Yaskawa INFORM job: DEMO_ROOF_SIDE_0625_3PAINT_24.JBI

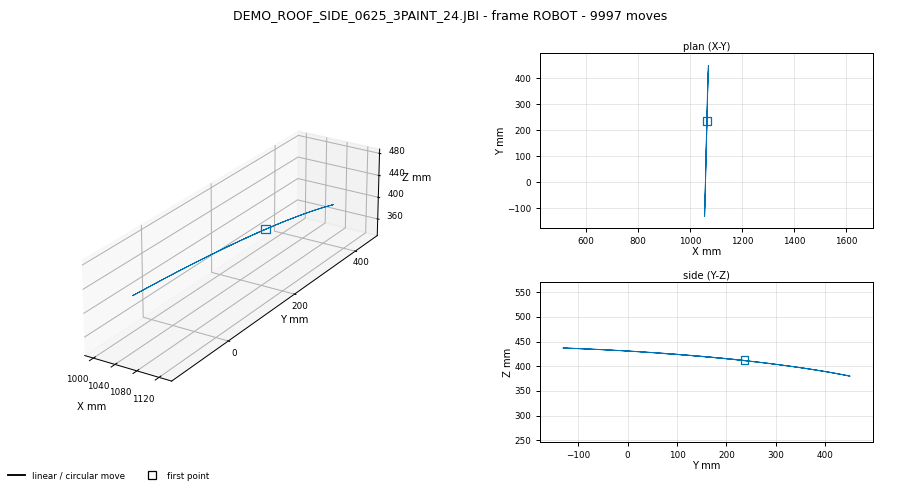
[picture p0: tool path of DEMO_ROOF_SIDE_0625_3PAINT_24.JBI in frame ROBOT, 9997 of 9997 moves have a stored position in this frame; points joined in program order, loops and branches not executed]
/JOB
//NAME DEMO_ROOF_SIDE_0625_3PAINT24
//POS
///NPOS 9997,0,0,0,0,0
///TOOL 0
///USER 0
///POSTYPE ROBOT
///RECTAN
///RCONF 1,0,0,0,0,0,0,0,0,0,0,0,0,0,0,0,0,0,0,0,0,0,0,0
C00000=1065.448,236.370,411.983,173.336,31.079,155.692
C00001=1065.443,236.150,412.007,173.335,31.075,155.691
C00002=1065.438,235.930,412.031,173.333,31.072,155.691
C00003=1065.433,235.710,412.055,173.331,31.069,155.690
C00004=1065.427,235.489,412.080,173.329,31.065,155.690
C00005=1065.422,235.270,412.102,173.326,31.062,155.689
C00006=1065.416,235.049,412.127,173.325,31.058,155.688
C00007=1065.411,234.830,412.151,173.323,31.055,155.688
C00008=1065.405,234.581,412.178,173.321,31.050,155.687
C00009=1065.399,234.332,412.204,173.318,31.047,155.686
C00010=1065.393,234.085,412.232,173.317,31.042,155.686
C00011=1065.388,233.835,412.259,173.314,31.038,155.685
C00012=1065.382,233.587,412.286,173.312,31.034,155.684
C00013=1065.376,233.339,412.313,173.309,31.030,155.683
C00014=1065.370,233.090,412.339,173.308,31.027,155.683
C00015=1065.364,232.842,412.367,173.305,31.022,155.682
C00016=1065.358,232.593,412.394,173.303,31.018,155.681
C00017=1065.352,232.345,412.420,173.300,31.015,155.681
C00018=1065.346,232.096,412.447,173.299,31.010,155.680
C00019=1065.340,231.848,412.474,173.296,31.006,155.679
C00020=1065.334,231.599,412.501,173.294,31.002,155.678
C00021=1065.328,231.350,412.528,173.293,30.998,155.678
C00022=1065.322,231.102,412.554,173.290,30.995,155.677
C00023=1065.316,230.853,412.581,173.288,30.990,155.676
C00024=1065.310,230.606,412.608,173.285,30.986,155.676
C00025=1065.304,230.357,412.635,173.284,30.982,155.675
C00026=1065.298,230.108,412.662,173.281,30.978,155.674
C00027=1065.292,229.860,412.689,173.279,30.975,155.674
C00028=1065.286,229.611,412.716,173.276,30.970,155.673
C00029=1065.280,229.363,412.742,173.275,30.966,155.672
C00030=1065.274,229.114,412.769,173.273,30.962,155.671
C00031=1065.268,228.866,412.794,173.270,30.958,155.671
C00032=1065.262,228.616,412.821,173.269,30.955,155.670
C00033=1065.256,228.368,412.848,173.266,30.950,155.669
C00034=1065.250,228.120,412.875,173.264,30.946,155.669
C00035=1065.244,227.871,412.902,173.261,30.943,155.668
C00036=1065.237,227.623,412.928,173.260,30.938,155.667
C00037=1065.232,227.374,412.954,173.258,30.935,155.667
C00038=1065.226,227.126,412.981,173.255,30.931,155.666
C00039=1065.220,226.878,413.008,173.253,30.926,155.665
C00040=1065.213,226.629,413.034,173.251,30.923,155.664
C00041=1065.207,226.380,413.060,173.249,30.919,155.664
C00042=1065.202,226.131,413.087,173.246,30.914,155.663
C00043=1065.196,225.883,413.113,173.245,30.911,155.662
C00044=1065.189,225.634,413.140,173.243,30.906,155.662
C00045=1065.183,225.386,413.166,173.240,30.903,155.661
C00046=1065.177,225.137,413.192,173.238,30.899,155.660
C00047=1065.172,224.889,413.219,173.236,30.894,155.659
C00048=1065.166,224.640,413.246,173.234,30.891,155.659
C00049=1065.159,224.392,413.272,173.232,30.886,155.658
C00050=1065.153,224.143,413.298,173.230,30.882,155.657
C00051=1065.148,223.894,413.325,173.228,30.878,155.657
C00052=1065.142,223.646,413.351,173.225,30.874,155.656
C00053=1065.135,223.398,413.377,173.223,30.870,155.655
C00054=1065.130,223.149,413.403,173.222,30.866,155.654
C00055=1065.124,222.900,413.430,173.219,30.862,155.654
C00056=1065.118,222.676,413.454,173.217,30.859,155.653
C00057=1065.113,222.452,413.477,173.215,30.855,155.652
C00058=1065.108,222.229,413.501,173.214,30.851,155.652
C00059=1065.102,222.004,413.525,173.212,30.848,155.651
C00060=1065.097,221.780,413.548,173.210,30.844,155.650
C00061=1065.092,221.556,413.572,173.208,30.841,155.650
C00062=1065.087,221.332,413.595,173.206,30.837,155.649
C00063=1065.080,221.108,413.619,173.204,30.833,155.649
C00064=1065.075,220.859,413.645,173.202,30.829,155.648
C00065=1065.069,220.611,413.671,173.200,30.825,155.647
C00066=1065.063,220.362,413.697,173.198,30.821,155.647
C00067=1065.057,220.114,413.723,173.196,30.817,155.646
C00068=1065.051,219.865,413.749,173.194,30.813,155.645
C00069=1065.044,219.616,413.775,173.192,30.809,155.644
C00070=1065.038,219.367,413.801,173.190,30.805,155.644
C00071=1065.032,219.119,413.827,173.187,30.801,155.643
C00072=1065.026,218.870,413.853,173.186,30.797,155.642
C00073=1065.020,218.622,413.879,173.184,30.793,155.642
C00074=1065.014,218.373,413.905,173.181,30.789,155.641
C00075=1065.008,218.125,413.931,173.180,30.785,155.640
C00076=1065.002,217.876,413.957,173.178,30.781,155.639
C00077=1064.996,217.628,413.983,173.175,30.777,155.639
C00078=1064.991,217.379,414.009,173.173,30.773,155.638
C00079=1064.984,217.131,414.034,173.172,30.769,155.637
C00080=1064.979,216.882,414.061,173.169,30.765,155.637
C00081=1064.972,216.634,414.086,173.167,30.760,155.636
C00082=1064.967,216.385,414.112,173.165,30.756,155.635
C00083=1064.960,216.137,414.138,173.163,30.752,155.634
C00084=1064.955,215.888,414.164,173.161,30.748,155.634
C00085=1064.949,215.639,414.190,173.160,30.744,155.633
C00086=1064.942,215.391,414.216,173.157,30.740,155.632
C00087=1064.937,215.142,414.242,173.155,30.736,155.631
C00088=1064.930,214.893,414.267,173.153,30.732,155.631
C00089=1064.925,214.645,414.294,173.151,30.728,155.630
C00090=1064.918,214.396,414.319,173.149,30.724,155.629
C00091=1064.913,214.147,414.345,173.147,30.720,155.629
C00092=1064.907,213.899,414.370,173.145,30.716,155.628
C00093=1064.900,213.651,414.396,173.143,30.712,155.627
C00094=1064.895,213.402,414.422,173.141,30.708,155.626
C00095=1064.889,213.153,414.448,173.139,30.703,155.626
C00096=1064.883,212.904,414.473,173.137,30.700,155.625
C00097=1064.877,212.655,414.499,173.135,30.695,155.624
C00098=1064.870,212.407,414.525,173.133,30.691,155.624
C00099=1064.864,212.159,414.550,173.131,30.687,155.623
C00100=1064.859,211.910,414.576,173.129,30.683,155.622
C00101=1064.853,211.662,414.601,173.127,30.679,155.621
C00102=1064.847,211.413,414.626,173.125,30.675,155.621
C00103=1064.842,211.164,414.652,173.123,30.671,155.620
C00104=1064.835,210.915,414.678,173.121,30.667,155.619
C00105=1064.829,210.667,414.703,173.119,30.663,155.619
C00106=1064.823,210.418,414.728,173.117,30.659,155.618
C00107=1064.817,210.169,414.754,173.115,30.655,155.617
C00108=1064.811,209.920,414.780,173.114,30.650,155.616
C00109=1064.805,209.672,414.805,173.111,30.646,155.616
C00110=1064.798,209.424,414.831,173.109,30.642,155.615
C00111=1064.792,209.175,414.856,173.108,30.638,155.614
C00112=1064.788,208.953,414.879,173.106,30.635,155.614
C00113=1064.782,208.732,414.901,173.104,30.631,155.613
C00114=1064.777,208.510,414.924,173.103,30.627,155.612
C00115=1064.771,208.288,414.947,173.101,30.624,155.612
C00116=1064.766,208.066,414.969,173.099,30.620,155.611
C00117=1064.761,207.845,414.992,173.097,30.616,155.610
C00118=1064.756,207.624,415.015,173.095,30.612,155.610
C00119=1064.750,207.401,415.037,173.093,30.609,155.609
C00120=1064.722,206.233,415.152,172.931,30.529,155.603
C00121=1064.714,205.844,415.190,172.928,30.523,155.602
C00122=1064.705,205.475,415.227,172.924,30.519,155.601
C00123=1064.696,205.104,415.263,172.922,30.514,155.601
C00124=1064.688,204.735,415.299,172.918,30.509,155.600
C00125=1064.679,204.365,415.336,172.915,30.504,155.599
C00126=1064.674,204.117,415.360,172.913,30.501,155.598
C00127=1064.668,203.867,415.385,172.910,30.498,155.598
C00128=1064.662,203.619,415.409,172.908,30.495,155.598
C00129=1064.656,203.370,415.434,172.906,30.492,155.597
C00130=1064.650,203.121,415.457,172.904,30.488,155.596
C00131=1064.645,202.873,415.482,172.901,30.485,155.596
C00132=1064.639,202.624,415.507,172.899,30.482,155.595
C00133=1064.634,202.375,415.531,172.897,30.479,155.595
C00134=1064.627,202.126,415.555,172.895,30.476,155.594
C00135=1064.622,201.878,415.579,172.892,30.472,155.594
C00136=1064.616,201.629,415.604,172.891,30.469,155.593
C00137=1064.610,201.380,415.628,172.888,30.466,155.593
C00138=1064.604,201.131,415.652,172.886,30.463,155.592
C00139=1064.598,200.883,415.676,172.883,30.460,155.592
C00140=1064.593,200.634,415.700,172.882,30.457,155.592
C00141=1064.586,200.385,415.724,172.880,30.454,155.591
C00142=1064.581,200.137,415.749,172.877,30.451,155.590
C00143=1064.574,199.888,415.773,172.875,30.448,155.590
C00144=1064.569,199.639,415.797,172.873,30.444,155.590
C00145=1064.562,199.390,415.821,172.871,30.441,155.589
C00146=1064.557,199.141,415.844,172.868,30.438,155.589
C00147=1064.551,198.893,415.868,172.867,30.435,155.588
C00148=1064.545,198.643,415.893,172.864,30.432,155.588
C00149=1064.539,198.395,415.916,172.862,30.429,155.587
C00150=1064.534,198.146,415.941,172.859,30.426,155.587
C00151=1064.527,197.897,415.965,172.858,30.423,155.586
C00152=1064.522,197.649,415.989,172.855,30.420,155.586
C00153=1064.515,197.400,416.013,172.853,30.417,155.585
C00154=1064.510,197.151,416.036,172.851,30.414,155.585
C00155=1064.504,196.902,416.060,172.849,30.411,155.584
C00156=1064.498,196.653,416.085,172.847,30.407,155.584
C00157=1064.492,196.405,416.108,172.844,30.405,155.583
C00158=1064.487,196.156,416.133,172.843,30.401,155.583
C00159=1064.481,195.907,416.156,172.840,30.398,155.582
C00160=1064.475,195.658,416.180,172.838,30.395,155.582
C00161=1064.469,195.410,416.204,172.836,30.392,155.581
C00162=1064.463,195.161,416.228,172.834,30.389,155.581
C00163=1064.458,194.912,416.251,172.832,30.386,155.580
C00164=1064.452,194.663,416.275,172.829,30.383,155.580
C00165=1064.446,194.415,416.299,172.827,30.380,155.579
C00166=1064.440,194.165,416.323,172.826,30.377,155.579
C00167=1064.435,193.917,416.347,172.823,30.373,155.578
C00168=1064.429,193.668,416.371,172.821,30.371,155.578
C00169=1064.423,193.419,416.394,172.819,30.367,155.577
C00170=1064.417,193.170,416.418,172.817,30.365,155.577
C00171=1064.411,192.922,416.442,172.815,30.362,155.576
C00172=1064.406,192.673,416.465,172.812,30.358,155.576
C00173=1064.400,192.424,416.489,172.811,30.355,155.576
C00174=1064.394,192.175,416.514,172.808,30.352,155.575
C00175=1064.388,191.926,416.537,172.806,30.349,155.574
C00176=1064.382,191.678,416.560,172.805,30.346,155.574
C00177=1064.377,191.429,416.584,172.802,30.343,155.574
C00178=1064.370,191.146,416.611,172.799,30.339,155.573
C00179=1064.364,190.863,416.638,172.797,30.336,155.572
C00180=1064.357,190.580,416.665,172.795,30.332,155.572
C00181=1064.351,190.297,416.692,172.792,30.329,155.571
C00182=1064.345,190.048,416.715,172.790,30.326,155.571
C00183=1064.340,189.799,416.739,172.789,30.323,155.570
C00184=1064.334,189.551,416.763,172.786,30.320,155.570
C00185=1064.328,189.301,416.786,172.784,30.317,155.569
C00186=1064.322,189.053,416.810,172.783,30.314,155.569
C00187=1064.316,188.804,416.833,172.780,30.311,155.569
C00188=1064.311,188.555,416.857,172.778,30.308,155.568
C00189=1064.305,188.306,416.880,172.776,30.304,155.567
C00190=1064.299,188.058,416.904,172.774,30.302,155.567
C00191=1064.294,187.809,416.927,172.772,30.298,155.567
C00192=1064.289,187.560,416.950,172.769,30.295,155.566
C00193=1064.282,187.311,416.974,172.767,30.292,155.566
C00194=1064.277,187.062,416.998,172.766,30.289,155.565
C00195=1064.271,186.814,417.022,172.763,30.286,155.565
C00196=1064.266,186.564,417.045,172.761,30.283,155.564
C00197=1064.260,186.315,417.068,172.760,30.280,155.564
C00198=1064.254,186.067,417.092,172.757,30.277,155.563
C00199=1064.249,185.818,417.115,172.755,30.274,155.563
C00200=1064.243,185.569,417.138,172.753,30.271,155.562
C00201=1064.237,185.321,417.162,172.752,30.268,155.562
C00202=1064.232,185.072,417.185,172.749,30.264,155.561
C00203=1064.227,184.823,417.208,172.747,30.262,155.561
C00204=1064.221,184.574,417.231,172.746,30.259,155.560
C00205=1064.214,184.325,417.255,172.743,30.256,155.560
C00206=1064.209,184.076,417.278,172.741,30.253,155.559
C00207=1064.203,183.827,417.301,172.739,30.250,155.559
C00208=1064.197,183.578,417.324,172.737,30.247,155.559
C00209=1064.191,183.330,417.348,172.735,30.244,155.558
C00210=1064.185,183.081,417.371,172.733,30.241,155.558
C00211=1064.179,182.831,417.394,172.731,30.238,155.557
C00212=1064.173,182.583,417.416,172.729,30.236,155.557
C00213=1064.167,182.334,417.439,172.727,30.232,155.556
C00214=1064.161,182.085,417.462,172.724,30.230,155.556
C00215=1064.155,181.836,417.485,172.723,30.227,155.555
C00216=1064.149,181.588,417.509,172.721,30.224,155.555
C00217=1064.144,181.339,417.532,172.718,30.221,155.554
C00218=1064.137,181.089,417.555,172.716,30.218,155.554
C00219=1064.131,180.841,417.578,172.715,30.215,155.554
C00220=1064.125,180.592,417.601,172.712,30.212,155.553
C00221=1064.119,180.343,417.623,172.710,30.209,155.553
C00222=1064.114,180.094,417.646,172.709,30.206,155.552
C00223=1064.108,179.845,417.669,172.706,30.203,155.552
C00224=1064.102,179.596,417.692,172.704,30.201,155.551
C00225=1064.096,179.347,417.715,172.702,30.198,155.551
C00226=1064.090,179.099,417.738,172.701,30.195,155.550
C00227=1064.084,178.850,417.761,172.698,30.192,155.550
C00228=1064.079,178.601,417.783,172.696,30.189,155.550
C00229=1064.073,178.352,417.806,172.695,30.186,155.549
C00230=1064.067,178.103,417.829,172.692,30.183,155.549
C00231=1064.061,177.854,417.852,172.690,30.180,155.548
C00232=1064.055,177.606,417.875,172.688,30.177,155.548
C00233=1064.049,177.357,417.898,172.687,30.175,155.547
C00234=1064.043,177.108,417.921,172.684,30.171,155.547
C00235=1064.038,176.859,417.944,172.682,30.169,155.546
C00236=1064.032,176.610,417.966,172.680,30.166,155.546
C00237=1064.025,176.362,417.989,172.679,30.163,155.545
C00238=1064.020,176.113,418.012,172.676,30.160,155.545
C00239=1064.014,175.864,418.035,172.674,30.157,155.545
C00240=1064.009,175.614,418.057,172.673,30.154,155.544
C00241=1064.003,175.365,418.080,172.670,30.151,155.544
C00242=1063.996,175.081,418.106,172.668,30.148,155.543
C00243=1063.989,174.798,418.132,172.666,30.144,155.543
C00244=1063.982,174.515,418.157,172.664,30.141,155.542
C00245=1063.975,174.232,418.183,172.661,30.138,155.542
C00246=1063.970,173.983,418.206,172.659,30.135,155.541
C00247=1063.964,173.734,418.229,172.658,30.132,155.541
C00248=1063.958,173.485,418.252,172.655,30.129,155.540
C00249=1063.953,173.236,418.274,172.653,30.126,155.540
C00250=1063.946,172.987,418.296,172.652,30.124,155.539
C00251=1063.941,172.739,418.319,172.650,30.120,155.539
C00252=1063.935,172.490,418.342,172.648,30.118,155.539
C00253=1063.930,172.240,418.364,172.645,30.115,155.538
C00254=1063.924,171.992,418.387,172.644,30.112,155.538
C00255=1063.918,171.743,418.410,172.642,30.109,155.537
C00256=1063.912,171.494,418.432,172.640,30.106,155.537
C00257=1063.907,171.245,418.455,172.638,30.103,155.536
C00258=1063.900,170.996,418.477,172.636,30.100,155.536
C00259=1063.895,170.747,418.500,172.634,30.098,155.535
C00260=1063.890,170.498,418.522,172.632,30.094,155.535
C00261=1063.884,170.249,418.545,172.631,30.092,155.534
C00262=1063.877,170.001,418.567,172.628,30.089,155.534
C00263=1063.872,169.751,418.589,172.626,30.086,155.534
C00264=1063.866,169.502,418.612,172.625,30.083,155.533
C00265=1063.860,169.254,418.635,172.623,30.080,155.533
C00266=1063.855,169.005,418.657,172.621,30.077,155.532
C00267=1063.849,168.756,418.679,172.618,30.074,155.532
C00268=1063.844,168.507,418.702,172.617,30.071,155.531
C00269=1063.837,168.258,418.724,172.615,30.068,155.531
C00270=1063.832,168.009,418.747,172.613,30.066,155.530
C00271=1063.827,167.760,418.769,172.612,30.063,155.530
C00272=1063.820,167.512,418.791,172.609,30.059,155.530
C00273=1063.815,167.262,418.813,172.607,30.057,155.529
C00274=1063.809,167.013,418.836,172.605,30.054,155.529
C00275=1063.804,166.764,418.859,172.604,30.051,155.528
C00276=1063.798,166.516,418.881,172.602,30.048,155.528
C00277=1063.793,166.266,418.903,172.599,30.045,155.527
C00278=1063.787,166.017,418.926,172.598,30.042,155.527
C00279=1063.781,165.768,418.947,172.596,30.039,155.526
C00280=1063.775,165.520,418.970,172.594,30.036,155.526
C00281=1063.770,165.271,418.992,172.592,30.033,155.525
C00282=1063.764,165.022,419.015,172.591,30.031,155.525
C00283=1063.758,164.772,419.037,172.588,30.027,155.525
C00284=1063.753,164.524,419.059,172.586,30.025,155.524
C00285=1063.747,164.275,419.081,172.585,30.022,155.524
C00286=1063.741,164.025,419.103,172.583,30.019,155.523
C00287=1063.736,163.777,419.126,172.581,30.016,155.523
C00288=1063.730,163.528,419.147,172.580,30.013,155.522
C00289=1063.724,163.279,419.170,172.577,30.010,155.522
C00290=1063.720,163.030,419.192,172.575,30.007,155.521
C00291=1063.713,162.781,419.214,172.573,30.004,155.521
C00292=1063.708,162.532,419.237,172.572,30.001,155.521
C00293=1063.703,162.283,419.259,172.570,29.999,155.520
C00294=1063.696,162.035,419.281,172.568,29.995,155.520
C00295=1063.691,161.785,419.303,172.567,29.993,155.519
C00296=1063.686,161.537,419.325,172.564,29.990,155.519
C00297=1063.680,161.288,419.348,172.562,29.987,155.518
C00298=1063.674,161.038,419.370,172.560,29.984,155.518
C00299=1063.668,160.789,419.391,172.559,29.981,155.517
C00300=1063.663,160.541,419.413,172.557,29.978,155.517
C00301=1063.657,160.292,419.436,172.555,29.975,155.516
C00302=1063.651,160.043,419.457,172.554,29.973,155.516
C00303=1063.645,159.794,419.479,172.551,29.970,155.516
C00304=1063.640,159.545,419.501,172.549,29.967,155.515
C00305=1063.634,159.295,419.522,172.548,29.964,155.515
C00306=1063.626,159.012,419.547,172.546,29.961,155.514
C00307=1063.620,158.728,419.572,172.543,29.958,155.514
C00308=1063.613,158.445,419.597,172.542,29.955,155.513
C00309=1063.607,158.161,419.622,172.539,29.952,155.513
C00310=1063.601,157.912,419.644,172.537,29.948,155.512
C00311=1063.596,157.663,419.666,172.535,29.946,155.512
C00312=1063.590,157.414,419.688,172.534,29.943,155.512
C00313=1063.584,157.165,419.709,172.532,29.940,155.511
C00314=1063.578,156.916,419.730,172.530,29.938,155.511
C00315=1063.573,156.667,419.753,172.529,29.934,155.510
C00316=1063.566,156.418,419.775,172.526,29.932,155.510
C00317=1063.561,156.170,419.796,172.524,29.929,155.509
C00318=1063.554,155.920,419.818,172.522,29.926,155.509
C00319=1063.549,155.671,419.840,172.521,29.923,155.509
C00320=1063.543,155.422,419.861,172.519,29.920,155.508
C00321=1063.537,155.173,419.883,172.517,29.918,155.508
C00322=1063.531,154.924,419.905,172.516,29.915,155.507
C00323=1063.526,154.675,419.927,172.514,29.912,155.507
C00324=1063.520,154.426,419.948,172.512,29.909,155.506
C00325=1063.514,154.177,419.970,172.509,29.907,155.506
C00326=1063.508,153.928,419.991,172.508,29.903,155.505
C00327=1063.502,153.679,420.013,172.506,29.901,155.505
C00328=1063.497,153.430,420.034,172.504,29.898,155.505
C00329=1063.490,153.181,420.056,172.503,29.895,155.504
C00330=1063.485,152.932,420.078,172.501,29.893,155.504
C00331=1063.480,152.683,420.099,172.499,29.890,155.503
C00332=1063.473,152.434,420.121,172.498,29.887,155.503
C00333=1063.468,152.186,420.142,172.496,29.884,155.502
C00334=1063.462,151.936,420.164,172.494,29.881,155.502
C00335=1063.456,151.686,420.185,172.491,29.878,155.502
C00336=1063.450,151.438,420.206,172.490,29.876,155.501
C00337=1063.445,151.188,420.228,172.488,29.873,155.501
C00338=1063.439,150.940,420.249,172.486,29.870,155.500
C00339=1063.433,150.691,420.271,172.485,29.867,155.500
C00340=1063.427,150.442,420.292,172.483,29.864,155.499
C00341=1063.421,150.193,420.314,172.481,29.862,155.499
C00342=1063.415,149.944,420.336,172.479,29.859,155.499
C00343=1063.410,149.695,420.356,172.478,29.856,155.498
C00344=1063.404,149.445,420.378,172.476,29.854,155.498
C00345=1063.398,149.197,420.399,172.474,29.851,155.497
C00346=1063.392,148.948,420.421,172.473,29.848,155.497
C00347=1063.386,148.699,420.442,172.471,29.845,155.496
C00348=1063.381,148.449,420.463,172.468,29.842,155.496
C00349=1063.375,148.201,420.484,172.467,29.839,155.496
C00350=1063.369,147.952,420.506,172.465,29.837,155.495
C00351=1063.363,147.703,420.527,172.463,29.834,155.495
C00352=1063.357,147.453,420.548,172.461,29.831,155.494
C00353=1063.351,147.204,420.570,172.460,29.829,155.494
C00354=1063.346,146.956,420.591,172.458,29.826,155.494
C00355=1063.340,146.707,420.613,172.456,29.823,155.493
C00356=1063.334,146.457,420.633,172.455,29.820,155.493
C00357=1063.328,146.208,420.655,172.453,29.817,155.492
C00358=1063.323,145.960,420.676,172.451,29.815,155.492
C00359=1063.317,145.710,420.697,172.449,29.812,155.491
C00360=1063.310,145.462,420.718,172.448,29.809,155.491
C00361=1063.304,145.212,420.739,172.446,29.806,155.491
C00362=1063.299,144.963,420.760,172.444,29.804,155.490
C00363=1063.293,144.714,420.781,172.442,29.801,155.490
C00364=1063.287,144.466,420.803,172.440,29.798,155.489
C00365=1063.281,144.216,420.824,172.438,29.795,155.489
C00366=1063.276,143.967,420.845,172.437,29.792,155.489
C00367=1063.270,143.717,420.866,172.435,29.790,155.488
C00368=1063.264,143.469,420.886,172.433,29.787,155.488
C00369=1063.258,143.220,420.908,172.431,29.784,155.487
C00370=1063.251,142.937,420.932,172.430,29.781,155.487
C00371=1063.245,142.653,420.956,172.428,29.778,155.486
C00372=1063.238,142.369,420.980,172.426,29.775,155.486
C00373=1063.231,142.085,421.004,172.424,29.771,155.485
C00374=1063.225,141.835,421.025,172.422,29.769,155.485
C00375=1063.220,141.586,421.046,172.420,29.766,155.485
C00376=1063.215,141.337,421.066,172.419,29.763,155.484
C00377=1063.208,141.088,421.088,172.417,29.761,155.484
C00378=1063.203,140.839,421.109,172.415,29.758,155.483
C00379=1063.196,140.590,421.130,172.414,29.755,155.483
C00380=1063.191,140.341,421.150,172.412,29.753,155.482
C00381=1063.185,140.092,421.172,172.410,29.750,155.482
C00382=1063.180,139.842,421.192,172.408,29.747,155.482
C00383=1063.174,139.593,421.213,172.407,29.744,155.481
C00384=1063.167,139.344,421.234,172.405,29.741,155.481
C00385=1063.162,139.095,421.255,172.403,29.738,155.480
C00386=1063.156,138.846,421.276,172.402,29.736,155.480
C00387=1063.150,138.597,421.296,172.400,29.733,155.479
C00388=1063.145,138.348,421.317,172.398,29.730,155.479
C00389=1063.139,138.099,421.338,172.397,29.728,155.479
C00390=1063.133,137.850,421.358,172.395,29.725,155.478
C00391=1063.126,137.601,421.380,172.393,29.722,155.478
C00392=1063.121,137.352,421.401,172.391,29.719,155.477
C00393=1063.115,137.103,421.420,172.389,29.717,155.477
C00394=1063.109,136.854,421.442,172.387,29.714,155.477
C00395=1063.104,136.605,421.463,172.385,29.711,155.476
C00396=1063.097,136.355,421.483,172.384,29.709,155.476
C00397=1063.092,136.107,421.504,172.382,29.706,155.475
C00398=1063.086,135.858,421.524,172.380,29.703,155.475
C00399=1063.080,135.608,421.545,172.379,29.700,155.475
C00400=1063.074,135.359,421.566,172.377,29.698,155.474
C00401=1063.068,135.111,421.586,172.375,29.695,155.474
C00402=1063.062,134.861,421.607,172.374,29.692,155.473
C00403=1063.056,134.612,421.627,172.372,29.689,155.473
C00404=1063.051,134.364,421.649,172.370,29.686,155.472
C00405=1063.045,134.114,421.669,172.368,29.684,155.472
C00406=1063.039,133.865,421.689,172.367,29.681,155.472
C00407=1063.034,133.616,421.710,172.365,29.678,155.471
C00408=1063.027,133.366,421.730,172.363,29.676,155.471
C00409=1063.022,133.118,421.752,172.363,29.673,155.470
C00410=1063.016,132.869,421.772,172.361,29.670,155.470
C00411=1063.010,132.619,421.792,172.359,29.668,155.470
C00412=1063.004,132.370,421.813,172.358,29.665,155.469
C00413=1062.998,132.121,421.833,172.356,29.662,155.469
C00414=1062.993,131.873,421.854,172.354,29.659,155.468
C00415=1062.986,131.623,421.875,172.352,29.657,155.468
C00416=1062.981,131.374,421.895,172.351,29.654,155.468
C00417=1062.974,131.125,421.915,172.349,29.651,155.467
C00418=1062.968,130.876,421.935,172.347,29.649,155.467
C00419=1062.963,130.627,421.956,172.346,29.646,155.466
C00420=1062.957,130.377,421.976,172.344,29.643,155.466
C00421=1062.951,130.128,421.996,172.342,29.641,155.465
C00422=1062.945,129.879,422.017,172.341,29.638,155.465
C00423=1062.939,129.630,422.037,172.339,29.635,155.465
C00424=1062.933,129.381,422.057,172.337,29.632,155.464
C00425=1062.928,129.132,422.078,172.335,29.630,155.464
C00426=1062.921,128.883,422.098,172.334,29.627,155.463
C00427=1062.915,128.634,422.119,172.332,29.624,155.463
C00428=1062.909,128.385,422.139,172.330,29.622,155.463
C00429=1062.903,128.136,422.159,172.329,29.619,155.462
C00430=1062.897,127.887,422.179,172.327,29.617,155.462
C00431=1062.891,127.638,422.199,172.325,29.614,155.462
C00432=1062.886,127.389,422.220,172.324,29.611,155.461
C00433=1062.880,127.140,422.240,172.322,29.609,155.461
C00434=1062.872,126.855,422.263,172.320,29.605,155.460
C00435=1062.866,126.571,422.286,172.318,29.602,155.460
C00436=1062.859,126.286,422.309,172.316,29.599,155.459
C00437=1062.853,126.003,422.332,172.314,29.596,155.459
C00438=1062.846,125.753,422.352,172.313,29.594,155.458
C00439=1062.840,125.504,422.372,172.311,29.591,155.458
C00440=1062.835,125.255,422.392,172.309,29.588,155.458
C00441=1062.829,125.006,422.412,172.307,29.586,155.457
C00442=1062.823,124.757,422.433,172.306,29.583,155.457
C00443=1062.817,124.508,422.453,172.304,29.580,155.456
C00444=1062.811,124.259,422.473,172.302,29.577,155.456
C00445=1062.805,124.010,422.493,172.301,29.575,155.456
C00446=1062.799,123.761,422.513,172.299,29.572,155.455
C00447=1062.793,123.511,422.533,172.297,29.569,155.455
C00448=1062.788,123.262,422.553,172.297,29.567,155.454
C00449=1062.782,123.013,422.573,172.295,29.564,155.454
C00450=1062.776,122.764,422.593,172.293,29.561,155.454
C00451=1062.770,122.515,422.613,172.292,29.559,155.453
C00452=1062.765,122.266,422.634,172.290,29.556,155.453
C00453=1062.758,122.016,422.653,172.288,29.553,155.452
C00454=1062.752,121.767,422.673,172.287,29.550,155.452
C00455=1062.746,121.518,422.693,172.285,29.548,155.452
C00456=1062.741,121.269,422.714,172.283,29.544,155.451
C00457=1062.735,121.020,422.733,172.281,29.542,155.451
C00458=1062.729,120.771,422.753,172.280,29.539,155.450
C00459=1062.723,120.522,422.773,172.278,29.536,155.450
C00460=1062.718,120.272,422.794,172.276,29.534,155.449
C00461=1062.712,120.023,422.813,172.275,29.531,155.449
C00462=1062.706,119.774,422.833,172.273,29.528,155.449
C00463=1062.700,119.525,422.853,172.272,29.526,155.448
C00464=1062.694,119.277,422.873,172.271,29.523,155.448
C00465=1062.689,119.027,422.893,172.269,29.520,155.447
C00466=1062.683,118.778,422.913,172.267,29.517,155.447
C00467=1062.677,118.529,422.933,172.266,29.515,155.447
C00468=1062.671,118.280,422.952,172.264,29.512,155.446
C00469=1062.665,118.031,422.972,172.262,29.509,155.446
C00470=1062.659,117.781,422.993,172.261,29.507,155.445
C00471=1062.654,117.532,423.012,172.259,29.504,155.445
C00472=1062.648,117.283,423.032,172.257,29.501,155.444
C00473=1062.642,117.033,423.051,172.256,29.498,155.444
C00474=1062.636,116.785,423.071,172.254,29.496,155.444
C00475=1062.631,116.536,423.092,172.253,29.493,155.443
C00476=1062.625,116.286,423.111,172.251,29.490,155.443
C00477=1062.619,116.037,423.131,172.250,29.488,155.442
C00478=1062.613,115.788,423.150,172.248,29.484,155.442
C00479=1062.607,115.539,423.170,172.246,29.482,155.441
C00480=1062.602,115.290,423.191,172.245,29.479,155.441
C00481=1062.596,115.040,423.210,172.243,29.476,155.441
C00482=1062.590,114.792,423.230,172.241,29.474,155.440
C00483=1062.585,114.542,423.249,172.240,29.471,155.440
C00484=1062.579,114.293,423.269,172.238,29.468,155.439
C00485=1062.573,114.044,423.288,172.236,29.465,155.439
C00486=1062.567,113.795,423.308,172.236,29.463,155.439
C00487=1062.561,113.546,423.328,172.234,29.460,155.438
C00488=1062.555,113.297,423.348,172.232,29.457,155.438
C00489=1062.550,113.048,423.367,172.231,29.455,155.437
C00490=1062.544,112.799,423.387,172.229,29.452,155.437
C00491=1062.538,112.549,423.406,172.227,29.449,155.437
C00492=1062.531,112.300,423.426,172.226,29.446,155.436
C00493=1062.526,112.050,423.446,172.224,29.444,155.436
C00494=1062.520,111.801,423.465,172.222,29.441,155.435
C00495=1062.514,111.552,423.485,172.221,29.438,155.435
C00496=1062.508,111.303,423.504,172.220,29.436,155.435
C00497=1062.502,111.054,423.524,172.218,29.433,155.434
C00498=1062.496,110.770,423.546,172.215,29.430,155.434
C00499=1062.488,110.485,423.568,172.214,29.427,155.433
C00500=1062.482,110.201,423.589,172.212,29.424,155.433
C00501=1062.475,109.917,423.612,172.211,29.421,155.432
C00502=1062.469,109.667,423.631,172.209,29.419,155.432
C00503=1062.463,109.419,423.651,172.207,29.416,155.432
C00504=1062.457,109.169,423.670,172.205,29.413,155.431
C00505=1062.451,108.920,423.689,172.204,29.410,155.431
C00506=1062.445,108.671,423.709,172.203,29.408,155.430
C00507=1062.439,108.422,423.728,172.201,29.405,155.430
C00508=1062.434,108.172,423.747,172.200,29.402,155.430
C00509=1062.428,107.924,423.767,172.198,29.400,155.429
C00510=1062.421,107.674,423.786,172.196,29.397,155.429
C00511=1062.416,107.425,423.805,172.195,29.394,155.428
C00512=1062.410,107.176,423.825,172.193,29.392,155.428
C00513=1062.404,106.927,423.845,172.191,29.389,155.428
C00514=1062.398,106.677,423.864,172.190,29.386,155.427
C00515=1062.392,106.428,423.882,172.189,29.384,155.427
C00516=1062.386,106.179,423.902,172.187,29.381,155.426
C00517=1062.381,105.931,423.921,172.186,29.378,155.426
C00518=1062.375,105.681,423.941,172.184,29.375,155.426
C00519=1062.369,105.432,423.959,172.182,29.373,155.425
C00520=1062.363,105.183,423.978,172.181,29.370,155.425
C00521=1062.357,104.933,423.998,172.179,29.368,155.424
C00522=1062.351,104.684,424.018,172.177,29.365,155.424
C00523=1062.345,104.435,424.036,172.176,29.362,155.424
C00524=1062.339,104.186,424.056,172.175,29.360,155.423
C00525=1062.333,103.936,424.075,172.173,29.357,155.423
C00526=1062.328,103.687,424.094,172.172,29.354,155.422
C00527=1062.321,103.438,424.113,172.170,29.352,155.422
C00528=1062.315,103.189,424.133,172.168,29.349,155.422
C00529=1062.310,102.940,424.152,172.167,29.346,155.421
C00530=1062.305,102.691,424.171,172.165,29.343,155.421
C00531=1062.298,102.442,424.189,172.164,29.341,155.420
C00532=1062.292,102.192,424.209,172.162,29.338,155.420
C00533=1062.287,101.943,424.228,172.161,29.335,155.420
C00534=1062.281,101.693,424.247,172.159,29.333,155.419
C00535=1062.275,101.444,424.266,172.157,29.330,155.419
C00536=1062.269,101.195,424.285,172.156,29.327,155.418
C00537=1062.263,100.945,424.304,172.154,29.324,155.418
C00538=1062.257,100.697,424.323,172.152,29.322,155.418
C00539=1062.252,100.448,424.342,172.152,29.319,155.417
C00540=1062.245,100.199,424.360,172.150,29.316,155.417
C00541=1062.240,99.949,424.380,172.148,29.314,155.416
C00542=1062.233,99.700,424.398,172.147,29.311,155.416
C00543=1062.228,99.451,424.418,172.145,29.309,155.416
C00544=1062.221,99.201,424.436,172.143,29.306,155.415
C00545=1062.215,98.952,424.455,172.142,29.303,155.415
C00546=1062.209,98.703,424.474,172.141,29.301,155.414
C00547=1062.204,98.454,424.493,172.139,29.298,155.414
C00548=1062.197,98.205,424.512,172.138,29.295,155.414
C00549=1062.192,97.956,424.531,172.136,29.293,155.413
C00550=1062.185,97.706,424.550,172.134,29.290,155.413
C00551=1062.180,97.457,424.569,172.133,29.287,155.412
C00552=1062.173,97.208,424.587,172.131,29.284,155.412
C00553=1062.168,96.958,424.607,172.129,29.282,155.412
C00554=1062.162,96.710,424.625,172.129,29.280,155.411
C00555=1062.156,96.461,424.644,172.127,29.277,155.411
C00556=1062.150,96.212,424.663,172.125,29.274,155.410
C00557=1062.144,95.961,424.681,172.124,29.271,155.410
C00558=1062.138,95.712,424.700,172.122,29.269,155.410
C00559=1062.132,95.463,424.719,172.120,29.266,155.409
C00560=1062.126,95.214,424.738,172.120,29.263,155.409
C00561=1062.121,94.965,424.757,172.118,29.261,155.408
C00562=1062.114,94.681,424.778,172.116,29.258,155.408
C00563=1062.107,94.396,424.800,172.114,29.254,155.407
C00564=1062.100,94.112,424.821,172.112,29.252,155.407
C00565=1062.094,93.828,424.842,172.110,29.248,155.407
C00566=1062.087,93.579,424.861,172.109,29.246,155.406
C00567=1062.082,93.330,424.879,172.108,29.243,155.406
C00568=1062.076,93.080,424.898,172.106,29.240,155.405
C00569=1062.069,92.831,424.916,172.105,29.238,155.405
C00570=1062.064,92.582,424.936,172.103,29.235,155.405
C00571=1062.058,92.333,424.954,172.101,29.233,155.404
C00572=1062.053,92.083,424.973,172.100,29.230,155.404
C00573=1062.046,91.834,424.991,172.098,29.227,155.403
C00574=1062.040,91.585,425.010,172.097,29.225,155.403
C00575=1062.035,91.336,425.029,172.096,29.222,155.403
C00576=1062.029,91.087,425.047,172.094,29.219,155.402
C00577=1062.023,90.837,425.066,172.092,29.216,155.402
C00578=1062.016,90.588,425.085,172.091,29.214,155.401
C00579=1062.011,90.339,425.102,172.089,29.211,155.401
C00580=1062.005,90.089,425.121,172.088,29.208,155.401
C00581=1061.999,89.840,425.140,172.087,29.206,155.400
C00582=1061.993,89.591,425.158,172.085,29.203,155.400
C00583=1061.987,89.342,425.176,172.083,29.201,155.399
C00584=1061.981,89.093,425.195,172.082,29.198,155.399
C00585=1061.975,88.843,425.213,172.080,29.195,155.399
C00586=1061.969,88.594,425.232,172.079,29.193,155.398
C00587=1061.963,88.345,425.250,172.078,29.190,155.398
C00588=1061.957,88.096,425.268,172.076,29.187,155.397
C00589=1061.951,87.846,425.287,172.074,29.185,155.397
C00590=1061.945,87.597,425.305,172.073,29.182,155.397
C00591=1061.939,87.348,425.324,172.071,29.180,155.396
C00592=1061.933,87.098,425.342,172.069,29.177,155.396
C00593=1061.926,86.849,425.360,172.069,29.174,155.396
C00594=1061.921,86.600,425.380,172.067,29.172,155.395
C00595=1061.915,86.351,425.397,172.065,29.169,155.395
C00596=1061.909,86.102,425.416,172.064,29.166,155.394
C00597=1061.903,85.852,425.434,172.062,29.164,155.394
C00598=1061.897,85.604,425.452,172.060,29.161,155.394
C00599=1061.891,85.354,425.470,172.060,29.159,155.393
C00600=1061.885,85.104,425.489,172.058,29.156,155.393
C00601=1061.880,84.855,425.507,172.056,29.153,155.392
C00602=1061.873,84.606,425.525,172.055,29.150,155.392
C00603=1061.867,84.356,425.543,172.053,29.148,155.392
C00604=1061.861,84.108,425.562,172.051,29.145,155.391
C00605=1061.855,83.858,425.580,172.051,29.143,155.391
C00606=1061.849,83.609,425.599,172.049,29.140,155.390
C00607=1061.844,83.360,425.616,172.047,29.137,155.390
C00608=1061.838,83.110,425.634,172.046,29.135,155.390
C00609=1061.831,82.861,425.653,172.044,29.132,155.389
C00610=1061.826,82.612,425.670,172.042,29.129,155.389
C00611=1061.819,82.363,425.689,172.042,29.127,155.388
C00612=1061.813,82.113,425.707,172.040,29.124,155.388
C00613=1061.808,81.864,425.726,172.038,29.121,155.388
C00614=1061.802,81.615,425.744,172.037,29.118,155.387
C00615=1061.797,81.366,425.761,172.035,29.116,155.387
C00616=1061.790,81.116,425.780,172.034,29.114,155.387
C00617=1061.784,80.867,425.798,172.033,29.111,155.386
C00618=1061.778,80.618,425.816,172.031,29.108,155.386
C00619=1061.772,80.369,425.834,172.029,29.105,155.385
C00620=1061.767,80.119,425.852,172.028,29.103,155.385
C00621=1061.761,79.870,425.871,172.026,29.100,155.385
C00622=1061.755,79.620,425.889,172.025,29.097,155.384
C00623=1061.749,79.371,425.907,172.024,29.095,155.384
C00624=1061.743,79.122,425.925,172.022,29.092,155.383
C00625=1061.737,78.873,425.943,172.020,29.089,155.383
C00626=1061.731,78.589,425.963,172.019,29.086,155.383
C00627=1061.724,78.305,425.984,172.017,29.083,155.382
C00628=1061.717,78.020,426.004,172.016,29.080,155.382
C00629=1061.710,77.735,426.025,172.014,29.077,155.381
C00630=1061.704,77.486,426.043,172.012,29.075,155.381
C00631=1061.698,77.237,426.061,172.011,29.072,155.380
C00632=1061.691,76.988,426.078,172.009,29.069,155.380
C00633=1061.686,76.739,426.096,172.008,29.067,155.380
C00634=1061.680,76.490,426.114,172.007,29.064,155.379
C00635=1061.674,76.241,426.132,172.005,29.062,155.379
C00636=1061.668,75.991,426.150,172.003,29.059,155.379
C00637=1061.662,75.741,426.168,172.002,29.056,155.378
C00638=1061.656,75.492,426.185,172.000,29.053,155.378
C00639=1061.650,75.243,426.204,171.999,29.051,155.377
C00640=1061.644,74.994,426.222,171.998,29.048,155.377
C00641=1061.638,74.744,426.240,171.996,29.046,155.377
C00642=1061.632,74.495,426.257,171.994,29.043,155.376
C00643=1061.626,74.246,426.274,171.993,29.040,155.376
C00644=1061.620,73.996,426.292,171.992,29.038,155.375
C00645=1061.614,73.747,426.310,171.990,29.035,155.375
C00646=1061.608,73.498,426.329,171.989,29.032,155.375
C00647=1061.602,73.249,426.346,171.987,29.030,155.374
C00648=1061.596,72.999,426.364,171.985,29.027,155.374
C00649=1061.590,72.750,426.381,171.984,29.025,155.374
C00650=1061.584,72.501,426.399,171.983,29.022,155.373
C00651=1061.578,72.251,426.417,171.981,29.019,155.373
C00652=1061.572,72.002,426.435,171.980,29.017,155.372
C00653=1061.567,71.753,426.452,171.978,29.014,155.372
C00654=1061.560,71.503,426.470,171.976,29.012,155.372
C00655=1061.555,71.254,426.488,171.976,29.009,155.371
C00656=1061.548,71.004,426.505,171.974,29.006,155.371
C00657=1061.543,70.755,426.523,171.972,29.004,155.370
C00658=1061.536,70.506,426.540,171.971,29.001,155.370
C00659=1061.531,70.257,426.558,171.969,28.998,155.370
C00660=1061.525,70.007,426.576,171.969,28.996,155.369
C00661=1061.519,69.758,426.593,171.967,28.993,155.369
C00662=1061.512,69.508,426.611,171.965,28.991,155.368
C00663=1061.507,69.259,426.628,171.964,28.988,155.368
C00664=1061.501,69.010,426.646,171.962,28.985,155.368
C00665=1061.495,68.761,426.663,171.960,28.982,155.367
C00666=1061.489,68.512,426.681,171.960,28.980,155.367
C00667=1061.483,68.262,426.699,171.958,28.978,155.367
C00668=1061.477,68.013,426.716,171.956,28.975,155.366
C00669=1061.471,67.764,426.734,171.955,28.972,155.366
C00670=1061.465,67.515,426.751,171.953,28.969,155.365
C00671=1061.458,67.265,426.769,171.952,28.967,155.365
C00672=1061.453,67.016,426.786,171.951,28.965,155.365
C00673=1061.446,66.766,426.804,171.949,28.962,155.364
C00674=1061.440,66.518,426.821,171.947,28.959,155.364
C00675=1061.434,66.267,426.838,171.946,28.956,155.363
C00676=1061.429,66.018,426.856,171.945,28.954,155.363
C00677=1061.423,65.770,426.873,171.943,28.952,155.363
C00678=1061.417,65.520,426.891,171.942,28.949,155.362
C00679=1061.411,65.271,426.908,171.940,28.946,155.362
C00680=1061.404,65.021,426.926,171.938,28.943,155.362
C00681=1061.399,64.772,426.943,171.937,28.940,155.361
C00682=1061.393,64.522,426.960,171.936,28.939,155.361
C00683=1061.387,64.273,426.977,171.934,28.936,155.360
C00684=1061.380,64.023,426.995,171.933,28.933,155.360
C00685=1061.374,63.775,427.012,171.931,28.930,155.360
C00686=1061.368,63.526,427.029,171.929,28.928,155.359
C00687=1061.362,63.276,427.047,171.929,28.925,155.359
C00688=1061.356,63.027,427.064,171.927,28.923,155.359
C00689=1061.350,62.777,427.081,171.925,28.921,155.358
C00690=1061.342,62.493,427.101,171.924,28.918,155.358
C00691=1061.336,62.209,427.120,171.922,28.914,155.357
C00692=1061.329,61.924,427.140,171.921,28.912,155.357
C00693=1061.322,61.640,427.160,171.919,28.909,155.357
C00694=1061.316,61.391,427.176,171.917,28.906,155.356
C00695=1061.310,61.141,427.194,171.916,28.903,155.356
C00696=1061.303,60.892,427.211,171.914,28.901,155.356
C00697=1061.297,60.643,427.228,171.912,28.898,155.355
C00698=1061.291,60.393,427.245,171.912,28.896,155.355
C00699=1061.285,60.144,427.262,171.910,28.894,155.354
C00700=1061.279,59.894,427.280,171.908,28.891,155.354
C00701=1061.273,59.645,427.296,171.907,28.888,155.354
C00702=1061.266,59.396,427.314,171.905,28.886,155.353
C00703=1061.261,59.147,427.331,171.903,28.883,155.353
C00704=1061.255,58.897,427.347,171.903,28.881,155.352
C00705=1061.248,58.648,427.365,171.901,28.878,155.352
C00706=1061.243,58.398,427.382,171.899,28.876,155.352
C00707=1061.236,58.149,427.399,171.898,28.873,155.351
C00708=1061.230,57.900,427.417,171.896,28.870,155.351
C00709=1061.224,57.650,427.433,171.895,28.868,155.351
C00710=1061.217,57.401,427.450,171.894,28.865,155.350
C00711=1061.212,57.151,427.467,171.892,28.863,155.350
C00712=1061.206,56.903,427.484,171.891,28.860,155.350
C00713=1061.199,56.653,427.501,171.889,28.858,155.349
C00714=1061.194,56.404,427.518,171.888,28.855,155.349
C00715=1061.188,56.155,427.535,171.887,28.852,155.348
C00716=1061.181,55.905,427.552,171.885,28.849,155.348
C00717=1061.176,55.656,427.569,171.883,28.847,155.348
C00718=1061.170,55.406,427.586,171.882,28.845,155.347
C00719=1061.163,55.157,427.603,171.880,28.842,155.347
C00720=1061.158,54.907,427.620,171.879,28.839,155.347
C00721=1061.151,54.659,427.637,171.878,28.837,155.346
C00722=1061.145,54.409,427.653,171.876,28.834,155.346
C00723=1061.139,54.159,427.671,171.874,28.831,155.345
C00724=1061.133,53.910,427.687,171.873,28.829,155.345
C00725=1061.127,53.661,427.704,171.872,28.827,155.345
C00726=1061.121,53.411,427.721,171.870,28.824,155.344
C00727=1061.115,53.162,427.738,171.869,28.821,155.344
C00728=1061.109,52.913,427.755,171.867,28.819,155.344
C00729=1061.104,52.663,427.771,171.866,28.816,155.343
C00730=1061.097,52.414,427.789,171.865,28.814,155.343
C00731=1061.091,52.164,427.805,171.863,28.811,155.342
C00732=1061.085,51.915,427.823,171.862,28.809,155.342
C00733=1061.079,51.666,427.839,171.860,28.806,155.342
C00734=1061.073,51.416,427.856,171.858,28.803,155.341
C00735=1061.067,51.167,427.873,171.858,28.801,155.341
C00736=1061.061,50.918,427.889,171.856,28.798,155.341
C00737=1061.055,50.669,427.906,171.854,28.796,155.340
C00738=1061.049,50.420,427.923,171.853,28.793,155.340
C00739=1061.043,50.169,427.940,171.851,28.790,155.340
C00740=1061.037,49.920,427.957,171.850,28.787,155.339
C00741=1061.031,49.671,427.973,171.849,28.785,155.339
C00742=1061.026,49.421,427.990,171.847,28.782,155.338
C00743=1061.020,49.173,428.007,171.845,28.780,155.338
C00744=1061.013,48.923,428.023,171.844,28.777,155.338
C00745=1061.007,48.673,428.040,171.843,28.775,155.337
C00746=1061.002,48.424,428.057,171.842,28.772,155.337
C00747=1060.996,48.175,428.074,171.840,28.769,155.337
C00748=1060.990,47.926,428.090,171.838,28.767,155.336
C00749=1060.983,47.676,428.107,171.837,28.764,155.336
C00750=1060.978,47.427,428.124,171.835,28.762,155.335
C00751=1060.972,47.177,428.140,171.834,28.759,155.335
C00752=1060.966,46.928,428.156,171.833,28.756,155.335
C00753=1060.960,46.679,428.174,171.831,28.753,155.334
C00754=1060.953,46.394,428.193,171.829,28.751,155.334
C00755=1060.947,46.110,428.212,171.828,28.748,155.333
C00756=1060.940,45.825,428.231,171.826,28.745,155.333
C00757=1060.933,45.541,428.249,171.825,28.742,155.333
C00758=1060.927,45.291,428.266,171.823,28.739,155.332
C00759=1060.921,45.041,428.283,171.821,28.737,155.332
C00760=1060.915,44.792,428.299,171.820,28.734,155.331
C00761=1060.909,44.543,428.316,171.819,28.731,155.331
C00762=1060.903,44.293,428.332,171.818,28.729,155.331
C00763=1060.898,44.044,428.349,171.816,28.726,155.330
C00764=1060.892,43.794,428.365,171.814,28.724,155.330
C00765=1060.886,43.545,428.382,171.813,28.721,155.330
C00766=1060.880,43.295,428.398,171.812,28.718,155.329
C00767=1060.874,43.046,428.414,171.810,28.716,155.329
C00768=1060.867,42.797,428.431,171.809,28.713,155.328
C00769=1060.861,42.548,428.448,171.807,28.711,155.328
C00770=1060.855,42.298,428.464,171.805,28.708,155.328
C00771=1060.849,42.049,428.480,171.805,28.706,155.327
C00772=1060.844,41.800,428.496,171.803,28.703,155.327
C00773=1060.838,41.550,428.513,171.801,28.701,155.327
C00774=1060.831,41.300,428.529,171.800,28.698,155.326
C00775=1060.825,41.051,428.546,171.798,28.695,155.326
C00776=1060.819,40.801,428.562,171.796,28.693,155.326
C00777=1060.813,40.552,428.578,171.796,28.690,155.325
C00778=1060.807,40.303,428.594,171.794,28.688,155.325
C00779=1060.801,40.053,428.611,171.793,28.685,155.324
C00780=1060.795,39.804,428.627,171.791,28.683,155.324
C00781=1060.789,39.555,428.643,171.789,28.680,155.324
C00782=1060.783,39.305,428.659,171.789,28.677,155.323
C00783=1060.777,39.056,428.676,171.787,28.675,155.323
C00784=1060.772,38.807,428.692,171.785,28.672,155.323
C00785=1060.766,38.557,428.708,171.784,28.670,155.322
C00786=1060.759,38.307,428.725,171.782,28.667,155.322
C00787=1060.753,38.058,428.741,171.781,28.665,155.322
C00788=1060.747,37.809,428.757,171.780,28.662,155.321
C00789=1060.741,37.559,428.774,171.778,28.660,155.321
C00790=1060.735,37.310,428.790,171.777,28.657,155.321
C00791=1060.729,37.061,428.806,171.775,28.655,155.320
C00792=1060.723,36.812,428.822,171.773,28.652,155.320
C00793=1060.717,36.562,428.838,171.773,28.649,155.319
C00794=1060.711,36.313,428.854,171.771,28.647,155.319
C00795=1060.705,36.063,428.871,171.769,28.644,155.319
C00796=1060.699,35.814,428.886,171.768,28.642,155.318
C00797=1060.692,35.564,428.902,171.766,28.639,155.318
C00798=1060.686,35.315,428.918,171.765,28.637,155.318
C00799=1060.680,35.065,428.935,171.764,28.635,155.317
C00800=1060.674,34.816,428.951,171.762,28.632,155.317
C00801=1060.668,34.566,428.967,171.760,28.630,155.317
C00802=1060.661,34.317,428.983,171.759,28.627,155.316
C00803=1060.656,34.067,428.998,171.757,28.625,155.316
C00804=1060.650,33.818,429.015,171.756,28.622,155.316
C00805=1060.644,33.569,429.031,171.755,28.619,155.315
C00806=1060.638,33.319,429.047,171.753,28.617,155.315
C00807=1060.631,33.070,429.063,171.752,28.614,155.315
C00808=1060.625,32.820,429.078,171.750,28.612,155.314
C00809=1060.619,32.571,429.095,171.749,28.609,155.314
C00810=1060.614,32.322,429.111,171.748,28.607,155.313
C00811=1060.607,32.073,429.126,171.746,28.604,155.313
C00812=1060.601,31.823,429.143,171.744,28.602,155.313
C00813=1060.595,31.573,429.158,171.743,28.599,155.313
C00814=1060.589,31.324,429.175,171.741,28.597,155.312
C00815=1060.583,31.075,429.190,171.740,28.595,155.312
C00816=1060.577,30.826,429.206,171.739,28.592,155.311
C00817=1060.571,30.576,429.222,171.737,28.589,155.311
C00818=1060.565,30.291,429.241,171.736,28.586,155.311
C00819=1060.558,30.007,429.258,171.734,28.584,155.310
C00820=1060.550,29.722,429.277,171.732,28.581,155.310
C00821=1060.544,29.437,429.294,171.731,28.578,155.309
C00822=1060.538,29.188,429.310,171.729,28.575,155.309
C00823=1060.532,28.938,429.326,171.728,28.573,155.309
C00824=1060.525,28.689,429.342,171.726,28.570,155.308
C00825=1060.519,28.440,429.358,171.724,28.568,155.308
C00826=1060.514,28.190,429.373,171.723,28.565,155.308
C00827=1060.507,27.941,429.389,171.722,28.563,155.307
C00828=1060.501,27.691,429.405,171.720,28.560,155.307
C00829=1060.495,27.441,429.421,171.719,28.558,155.307
C00830=1060.489,27.192,429.437,171.717,28.555,155.306
C00831=1060.483,26.942,429.452,171.715,28.553,155.306
C00832=1060.476,26.693,429.468,171.715,28.551,155.306
C00833=1060.470,26.444,429.484,171.713,28.548,155.305
C00834=1060.464,26.194,429.499,171.711,28.546,155.305
C00835=1060.459,25.946,429.515,171.710,28.543,155.305
C00836=1060.453,25.696,429.530,171.708,28.541,155.304
C00837=1060.446,25.447,429.546,171.707,28.538,155.304
C00838=1060.441,25.197,429.562,171.706,28.536,155.304
C00839=1060.434,24.948,429.577,171.704,28.534,155.303
C00840=1060.428,24.698,429.593,171.703,28.531,155.303
C00841=1060.422,24.449,429.608,171.701,28.528,155.303
C00842=1060.416,24.199,429.624,171.699,28.526,155.302
C00843=1060.409,23.950,429.640,171.698,28.523,155.302
C00844=1060.404,23.700,429.655,171.697,28.521,155.302
C00845=1060.397,23.451,429.671,171.695,28.519,155.301
C00846=1060.392,23.201,429.686,171.694,28.516,155.301
C00847=1060.385,22.952,429.702,171.692,28.514,155.301
C00848=1060.380,22.702,429.717,171.690,28.511,155.300
C00849=1060.373,22.453,429.733,171.689,28.509,155.300
C00850=1060.367,22.203,429.748,171.688,28.506,155.300
C00851=1060.361,21.954,429.764,171.686,28.504,155.299
C00852=1060.355,21.704,429.780,171.685,28.501,155.299
C00853=1060.348,21.455,429.795,171.683,28.499,155.299
C00854=1060.343,21.206,429.811,171.682,28.496,155.298
C00855=1060.337,20.956,429.825,171.680,28.494,155.298
C00856=1060.331,20.707,429.842,171.679,28.491,155.298
C00857=1060.324,20.457,429.857,171.678,28.489,155.297
C00858=1060.319,20.208,429.873,171.676,28.486,155.297
C00859=1060.312,19.958,429.888,171.674,28.484,155.297
C00860=1060.307,19.709,429.903,171.673,28.481,155.296
C00861=1060.300,19.460,429.919,171.671,28.479,155.296
C00862=1060.294,19.210,429.934,171.670,28.476,155.296
C00863=1060.288,18.961,429.949,171.669,28.474,155.295
C00864=1060.282,18.711,429.965,171.667,28.472,155.295
C00865=1060.276,18.462,429.980,171.666,28.469,155.295
C00866=1060.270,18.212,429.995,171.664,28.467,155.294
C00867=1060.264,17.964,430.011,171.662,28.464,155.294
C00868=1060.258,17.714,430.026,171.661,28.462,155.294
C00869=1060.252,17.464,430.041,171.660,28.459,155.293
C00870=1060.245,17.215,430.057,171.658,28.457,155.293
C00871=1060.239,16.965,430.072,171.657,28.455,155.293
C00872=1060.233,16.716,430.087,171.655,28.452,155.292
C00873=1060.228,16.466,430.102,171.653,28.450,155.292
C00874=1060.221,16.217,430.118,171.652,28.447,155.292
C00875=1060.215,15.967,430.133,171.651,28.445,155.291
C00876=1060.209,15.717,430.149,171.650,28.442,155.291
C00877=1060.203,15.468,430.163,171.648,28.440,155.291
C00878=1060.197,15.219,430.179,171.646,28.438,155.290
C00879=1060.191,14.969,430.194,171.645,28.435,155.290
C00880=1060.185,14.720,430.209,171.643,28.433,155.290
C00881=1060.179,14.471,430.224,171.641,28.430,155.289
C00882=1060.172,14.187,430.242,171.640,28.427,155.289
C00883=1060.164,13.903,430.258,171.638,28.425,155.289
C00884=1060.158,13.620,430.276,171.637,28.422,155.288
C00885=1060.150,13.337,430.293,171.635,28.419,155.288
C00886=1060.144,13.088,430.308,171.633,28.417,155.288
C00887=1060.138,12.838,430.323,171.632,28.415,155.287
C00888=1060.133,12.589,430.338,171.630,28.412,155.287
C00889=1060.126,12.339,430.353,171.629,28.410,155.287
C00890=1060.120,12.089,430.368,171.628,28.408,155.286
C00891=1060.113,11.840,430.383,171.626,28.405,155.286
C00892=1060.107,11.591,430.399,171.624,28.403,155.286
C00893=1060.101,11.342,430.413,171.623,28.401,155.285
C00894=1060.095,11.092,430.428,171.621,28.398,155.285
C00895=1060.088,10.843,430.443,171.619,28.396,155.285
C00896=1060.083,10.593,430.459,171.619,28.394,155.285
C00897=1060.077,10.344,430.473,171.617,28.391,155.284
C00898=1060.070,10.094,430.488,171.616,28.389,155.284
C00899=1060.064,9.844,430.503,171.614,28.386,155.284
C00900=1060.058,9.595,430.518,171.612,28.384,155.283
C00901=1060.052,9.346,430.533,171.611,28.381,155.283
C00902=1060.046,9.096,430.548,171.609,28.379,155.283
C00903=1060.039,8.846,430.562,171.608,28.377,155.282
C00904=1060.033,8.597,430.577,171.607,28.375,155.282
C00905=1060.027,8.348,430.592,171.605,28.372,155.282
C00906=1060.021,8.098,430.607,171.603,28.370,155.281
C00907=1060.015,7.848,430.622,171.602,28.368,155.281
C00908=1060.009,7.599,430.637,171.600,28.365,155.281
C00909=1060.003,7.349,430.652,171.598,28.362,155.280
C00910=1059.996,7.100,430.667,171.597,28.360,155.280
C00911=1059.991,6.851,430.682,171.596,28.358,155.280
C00912=1059.984,6.601,430.696,171.594,28.355,155.280
C00913=1059.978,6.352,430.711,171.593,28.353,155.279
C00914=1059.972,6.103,430.726,171.591,28.351,155.279
C00915=1059.966,5.853,430.741,171.590,28.348,155.279
C00916=1059.959,5.603,430.756,171.588,28.346,155.278
C00917=1059.954,5.354,430.770,171.586,28.344,155.278
C00918=1059.947,5.104,430.785,171.586,28.342,155.278
C00919=1059.941,4.854,430.800,171.584,28.339,155.277
C00920=1059.935,4.605,430.814,171.582,28.337,155.277
C00921=1059.930,4.355,430.830,171.581,28.334,155.277
C00922=1059.923,4.106,430.845,171.579,28.332,155.276
C00923=1059.917,3.857,430.859,171.577,28.329,155.276
C00924=1059.911,3.607,430.874,171.576,28.327,155.276
C00925=1059.906,3.358,430.888,171.574,28.325,155.276
C00926=1059.899,3.108,430.903,171.573,28.322,155.275
C00927=1059.893,2.858,430.918,171.572,28.320,155.275
C00928=1059.887,2.609,430.933,171.570,28.318,155.275
C00929=1059.881,2.360,430.948,171.568,28.316,155.274
C00930=1059.875,2.111,430.962,171.567,28.313,155.274
C00931=1059.869,1.860,430.976,171.565,28.311,155.274
C00932=1059.862,1.611,430.991,171.564,28.308,155.273
C00933=1059.857,1.362,431.006,171.562,28.306,155.273
C00934=1059.850,1.112,431.021,171.561,28.304,155.273
C00935=1059.845,0.863,431.035,171.560,28.301,155.272
C00936=1059.838,0.613,431.050,171.558,28.299,155.272
C00937=1059.833,0.364,431.064,171.556,28.296,155.272
C00938=1059.826,0.114,431.079,171.555,28.294,155.272
C00939=1059.821,-0.135,431.093,171.553,28.292,155.271
C00940=1059.814,-0.385,431.108,171.551,28.290,155.271
C00941=1059.808,-0.635,431.123,171.550,28.287,155.271
C00942=1059.802,-0.883,431.137,171.549,28.285,155.270
C00943=1059.796,-1.134,431.152,171.548,28.283,155.270
C00944=1059.790,-1.383,431.166,171.546,28.280,155.270
C00945=1059.784,-1.632,431.181,171.544,28.277,155.269
C00946=1059.778,-1.914,431.198,171.543,28.275,155.269
C00947=1059.771,-2.195,431.213,171.541,28.272,155.269
C00948=1059.764,-2.477,431.230,171.540,28.270,155.268
C00949=1059.757,-2.758,431.246,171.537,28.267,155.268
C00950=1059.751,-3.007,431.260,171.536,28.265,155.268
C00951=1059.745,-3.257,431.275,171.535,28.262,155.267
C00952=1059.739,-3.506,431.290,171.533,28.260,155.267
C00953=1059.733,-3.756,431.304,171.531,28.258,155.267
C00954=1059.727,-4.006,431.319,171.530,28.256,155.267
C00955=1059.721,-4.255,431.332,171.528,28.253,155.266
C00956=1059.714,-4.505,431.347,171.526,28.251,155.266
C00957=1059.709,-4.754,431.361,171.525,28.248,155.266
C00958=1059.702,-5.003,431.375,171.523,28.246,155.265
C00959=1059.696,-5.252,431.390,171.522,28.244,155.265
C00960=1059.690,-5.503,431.404,171.521,28.242,155.265
C00961=1059.684,-5.752,431.419,171.519,28.240,155.265
C00962=1059.677,-6.002,431.433,171.517,28.237,155.264
C00963=1059.671,-6.251,431.447,171.516,28.235,155.264
C00964=1059.665,-6.501,431.461,171.514,28.233,155.264
C00965=1059.658,-6.750,431.476,171.513,28.231,155.263
C00966=1059.653,-7.000,431.490,171.511,28.228,155.263
C00967=1059.646,-7.249,431.504,171.509,28.226,155.263
C00968=1059.640,-7.499,431.518,171.508,28.224,155.263
C00969=1059.634,-7.748,431.532,171.506,28.222,155.262
C00970=1059.628,-7.998,431.547,171.505,28.220,155.262
C00971=1059.622,-8.247,431.561,171.504,28.217,155.262
C00972=1059.616,-8.497,431.575,171.502,28.215,155.261
C00973=1059.610,-8.746,431.589,171.500,28.212,155.261
C00974=1059.604,-8.996,431.604,171.499,28.210,155.261
C00975=1059.598,-9.245,431.617,171.497,28.208,155.261
C00976=1059.591,-9.495,431.632,171.495,28.206,155.260
C00977=1059.586,-9.745,431.646,171.494,28.203,155.260
C00978=1059.579,-9.994,431.660,171.492,28.201,155.260
C00979=1059.573,-10.244,431.674,171.490,28.199,155.260
C00980=1059.567,-10.493,431.689,171.490,28.197,155.259
C00981=1059.560,-10.742,431.702,171.488,28.195,155.259
C00982=1059.555,-10.992,431.716,171.486,28.192,155.259
C00983=1059.549,-11.242,431.731,171.485,28.190,155.258
C00984=1059.542,-11.491,431.744,171.483,28.188,155.258
C00985=1059.536,-11.741,431.758,171.481,28.186,155.258
C00986=1059.531,-11.990,431.773,171.480,28.183,155.258
C00987=1059.524,-12.239,431.786,171.478,28.181,155.257
C00988=1059.518,-12.490,431.800,171.477,28.179,155.257
C00989=1059.512,-12.738,431.814,171.475,28.177,155.257
C00990=1059.506,-12.989,431.829,171.473,28.175,155.257
C00991=1059.500,-13.238,431.843,171.472,28.172,155.256
C00992=1059.494,-13.487,431.857,171.471,28.170,155.256
C00993=1059.488,-13.737,431.871,171.469,28.167,155.256
C00994=1059.482,-13.987,431.885,171.468,28.165,155.255
C00995=1059.475,-14.236,431.899,171.466,28.163,155.255
C00996=1059.469,-14.486,431.913,171.464,28.161,155.255
C00997=1059.463,-14.735,431.926,171.463,28.158,155.255
C00998=1059.457,-14.985,431.940,171.461,28.156,155.254
C00999=1059.451,-15.234,431.955,171.459,28.154,155.254
C01000=1059.445,-15.483,431.968,171.458,28.152,155.254
C01001=1059.438,-15.733,431.982,171.456,28.150,155.254
C01002=1059.433,-15.983,431.996,171.454,28.148,155.253
C01003=1059.426,-16.233,432.009,171.453,28.146,155.253
C01004=1059.420,-16.482,432.024,171.452,28.144,155.253
C01005=1059.414,-16.731,432.037,171.450,28.141,155.252
C01006=1059.408,-16.981,432.051,171.449,28.139,155.252
C01007=1059.402,-17.231,432.065,171.447,28.137,155.252
C01008=1059.396,-17.480,432.078,171.446,28.135,155.252
C01009=1059.390,-17.730,432.092,171.444,28.133,155.252
C01010=1059.382,-18.010,432.108,171.442,28.130,155.251
C01011=1059.376,-18.289,432.124,171.441,28.128,155.251
C01012=1059.368,-18.569,432.139,171.438,28.125,155.251
C01013=1059.361,-18.849,432.154,171.436,28.123,155.250
C01014=1059.356,-19.099,432.168,171.435,28.121,155.250
C01015=1059.349,-19.348,432.181,171.433,28.119,155.250
C01016=1059.343,-19.598,432.195,171.431,28.116,155.250
C01017=1059.337,-19.847,432.209,171.430,28.114,155.249
C01018=1059.331,-20.097,432.222,171.429,28.112,155.249
C01019=1059.325,-20.346,432.236,171.427,28.110,155.249
C01020=1059.319,-20.596,432.249,171.426,28.108,155.249
C01021=1059.312,-20.845,432.263,171.424,28.106,155.248
C01022=1059.307,-21.094,432.277,171.422,28.104,155.248
C01023=1059.300,-21.344,432.291,171.421,28.102,155.248
C01024=1059.294,-21.594,432.305,171.419,28.099,155.248
C01025=1059.288,-21.843,432.318,171.417,28.097,155.247
C01026=1059.281,-22.093,432.332,171.416,28.095,155.247
C01027=1059.276,-22.343,432.346,171.414,28.093,155.247
C01028=1059.270,-22.592,432.359,171.412,28.091,155.247
C01029=1059.263,-22.841,432.372,171.411,28.089,155.246
C01030=1059.257,-23.091,432.386,171.409,28.086,155.246
C01031=1059.251,-23.341,432.400,171.408,28.084,155.246
C01032=1059.245,-23.590,432.413,171.406,28.082,155.246
C01033=1059.239,-23.840,432.427,171.404,28.080,155.245
C01034=1059.233,-24.090,432.440,171.403,28.078,155.245
C01035=1059.226,-24.339,432.454,171.402,28.076,155.245
C01036=1059.221,-24.589,432.467,171.400,28.074,155.245
C01037=1059.215,-24.838,432.480,171.399,28.071,155.244
C01038=1059.209,-25.088,432.493,171.397,28.070,155.244
C01039=1059.203,-25.338,432.508,171.395,28.068,155.244
C01040=1059.196,-25.587,432.521,171.394,28.065,155.244
C01041=1059.190,-25.836,432.534,171.392,28.063,155.243
C01042=1059.185,-26.086,432.548,171.390,28.061,155.243
C01043=1059.179,-26.335,432.561,171.389,28.059,155.243
C01044=1059.172,-26.585,432.575,171.387,28.057,155.243
C01045=1059.166,-26.835,432.589,171.385,28.055,155.242
C01046=1059.160,-27.085,432.601,171.384,28.052,155.242
C01047=1059.154,-27.334,432.615,171.382,28.051,155.242
C01048=1059.147,-27.584,432.628,171.380,28.048,155.242
C01049=1059.141,-27.833,432.641,171.379,28.046,155.241
C01050=1059.135,-28.082,432.655,171.377,28.045,155.241
C01051=1059.129,-28.332,432.668,171.375,28.042,155.241
C01052=1059.124,-28.582,432.681,171.374,28.040,155.241
C01053=1059.117,-28.832,432.695,171.372,28.038,155.241
C01054=1059.110,-29.081,432.708,171.370,28.036,155.240
C01055=1059.104,-29.330,432.721,171.369,28.034,155.240
C01056=1059.098,-29.580,432.735,171.367,28.032,155.240
C01057=1059.092,-29.829,432.747,171.365,28.030,155.240
C01058=1059.085,-30.079,432.761,171.365,28.028,155.239
C01059=1059.079,-30.329,432.774,171.363,28.026,155.239
C01060=1059.073,-30.578,432.787,171.361,28.024,155.239
C01061=1059.067,-30.828,432.800,171.360,28.022,155.239
C01062=1059.062,-31.077,432.814,171.358,28.020,155.238
C01063=1059.055,-31.327,432.827,171.356,28.018,155.238
C01064=1059.049,-31.577,432.840,171.354,28.016,155.238
C01065=1059.043,-31.827,432.853,171.353,28.014,155.238
C01066=1059.036,-32.076,432.866,171.351,28.012,155.238
C01067=1059.030,-32.325,432.880,171.349,28.010,155.237
C01068=1059.024,-32.575,432.892,171.348,28.008,155.237
C01069=1059.018,-32.824,432.906,171.346,28.006,155.237
C01070=1059.012,-33.073,432.919,171.344,28.004,155.237
C01071=1059.005,-33.324,432.932,171.343,28.002,155.236
C01072=1058.999,-33.573,432.945,171.341,28.000,155.236
C01073=1058.993,-33.823,432.958,171.339,27.998,155.236
C01074=1058.986,-34.102,432.973,171.338,27.995,155.236
C01075=1058.980,-34.381,432.988,171.336,27.993,155.235
C01076=1058.973,-34.660,433.002,171.334,27.991,155.235
C01077=1058.966,-34.939,433.016,171.332,27.988,155.235
C01078=1058.960,-35.188,433.029,171.330,27.987,155.235
C01079=1058.954,-35.438,433.043,171.329,27.984,155.235
C01080=1058.948,-35.688,433.055,171.327,27.983,155.234
C01081=1058.941,-35.937,433.068,171.325,27.981,155.234
C01082=1058.936,-36.187,433.082,171.324,27.978,155.234
C01083=1058.930,-36.436,433.095,171.322,27.977,155.234
C01084=1058.924,-36.686,433.108,171.320,27.974,155.233
C01085=1058.917,-36.936,433.121,171.319,27.973,155.233
C01086=1058.911,-37.185,433.134,171.317,27.970,155.233
C01087=1058.905,-37.435,433.147,171.315,27.969,155.233
C01088=1058.899,-37.685,433.160,171.314,27.967,155.233
C01089=1058.893,-37.934,433.173,171.312,27.964,155.232
C01090=1058.887,-38.184,433.186,171.310,27.963,155.232
C01091=1058.881,-38.434,433.198,171.309,27.960,155.232
C01092=1058.875,-38.683,433.212,171.307,27.959,155.232
C01093=1058.869,-38.933,433.224,171.305,27.956,155.232
C01094=1058.862,-39.182,433.237,171.304,27.955,155.231
C01095=1058.856,-39.432,433.250,171.302,27.953,155.231
C01096=1058.850,-39.681,433.262,171.300,27.951,155.231
C01097=1058.844,-39.931,433.275,171.298,27.949,155.231
C01098=1058.838,-40.181,433.288,171.298,27.947,155.231
C01099=1058.831,-40.429,433.301,171.296,27.945,155.230
C01100=1058.825,-40.679,433.313,171.294,27.943,155.230
C01101=1058.819,-40.929,433.326,171.293,27.942,155.230
C01102=1058.813,-41.179,433.339,171.291,27.940,155.230
C01103=1058.807,-41.428,433.352,171.289,27.938,155.230
C01104=1058.800,-41.677,433.364,171.288,27.936,155.229
C01105=1058.794,-41.927,433.377,171.286,27.934,155.229
C01106=1058.788,-42.177,433.390,171.284,27.932,155.229
C01107=1058.782,-42.426,433.403,171.283,27.930,155.229
C01108=1058.776,-42.676,433.415,171.281,27.928,155.229
C01109=1058.769,-42.925,433.428,171.279,27.926,155.228
C01110=1058.763,-43.175,433.440,171.277,27.925,155.228
C01111=1058.757,-43.425,433.453,171.276,27.922,155.228
C01112=1058.751,-43.674,433.466,171.274,27.921,155.228
C01113=1058.745,-43.924,433.479,171.272,27.919,155.228
C01114=1058.739,-44.174,433.491,171.271,27.917,155.227
C01115=1058.733,-44.424,433.503,171.269,27.915,155.227
C01116=1058.726,-44.673,433.517,171.267,27.913,155.227
C01117=1058.721,-44.923,433.529,171.266,27.911,155.227
C01118=1058.714,-45.172,433.541,171.264,27.910,155.227
C01119=1058.708,-45.422,433.554,171.262,27.907,155.227
C01120=1058.702,-45.671,433.567,171.261,27.906,155.226
C01121=1058.696,-45.921,433.579,171.259,27.904,155.226
C01122=1058.689,-46.171,433.591,171.256,27.902,155.226
C01123=1058.683,-46.420,433.605,171.255,27.900,155.226
C01124=1058.677,-46.670,433.617,171.253,27.898,155.226
C01125=1058.671,-46.920,433.630,171.251,27.896,155.225
C01126=1058.665,-47.170,433.642,171.250,27.894,155.225
C01127=1058.659,-47.419,433.654,171.248,27.893,155.225
C01128=1058.653,-47.668,433.667,171.246,27.890,155.225
C01129=1058.647,-47.918,433.680,171.244,27.889,155.225
C01130=1058.640,-48.167,433.692,171.243,27.887,155.225
C01131=1058.635,-48.417,433.704,171.241,27.885,155.224
C01132=1058.629,-48.667,433.717,171.239,27.883,155.224
C01133=1058.622,-48.916,433.730,171.238,27.881,155.224
C01134=1058.616,-49.166,433.742,171.236,27.880,155.224
C01135=1058.610,-49.416,433.755,171.234,27.877,155.224
C01136=1058.604,-49.666,433.767,171.233,27.876,155.223
C01137=1058.598,-49.915,433.779,171.231,27.874,155.223
C01138=1058.591,-50.194,433.793,171.229,27.872,155.223
C01139=1058.584,-50.474,433.807,171.228,27.870,155.223
C01140=1058.577,-50.753,433.820,171.226,27.868,155.223
C01141=1058.570,-51.033,433.835,171.223,27.866,155.223
C01142=1058.564,-51.282,433.847,171.222,27.864,155.222
C01143=1058.557,-51.532,433.859,171.220,27.863,155.222
C01144=1058.551,-51.782,433.871,171.218,27.861,155.222
C01145=1058.544,-52.031,433.883,171.216,27.859,155.222
C01146=1058.539,-52.281,433.895,171.215,27.858,155.222
C01147=1058.533,-52.530,433.907,171.213,27.856,155.222
C01148=1058.527,-52.780,433.920,171.211,27.854,155.222
C01149=1058.520,-53.030,433.932,171.210,27.853,155.221
C01150=1058.513,-53.279,433.944,171.208,27.850,155.221
C01151=1058.507,-53.529,433.956,171.206,27.849,155.221
C01152=1058.501,-53.779,433.968,171.205,27.847,155.221
C01153=1058.495,-54.029,433.981,171.203,27.845,155.221
C01154=1058.488,-54.278,433.993,171.201,27.844,155.221
C01155=1058.482,-54.527,434.004,171.199,27.842,155.220
C01156=1058.476,-54.777,434.017,171.198,27.840,155.220
C01157=1058.470,-55.026,434.029,171.196,27.839,155.220
C01158=1058.464,-55.276,434.042,171.194,27.837,155.220
C01159=1058.457,-55.526,434.054,171.192,27.835,155.220
C01160=1058.450,-55.775,434.065,171.191,27.834,155.220
C01161=1058.444,-56.025,434.078,171.189,27.832,155.220
C01162=1058.439,-56.275,434.089,171.187,27.830,155.219
C01163=1058.433,-56.525,434.101,171.186,27.828,155.219
C01164=1058.426,-56.774,434.113,171.184,27.827,155.219
C01165=1058.420,-57.024,434.125,171.182,27.825,155.219
C01166=1058.414,-57.274,434.138,171.180,27.823,155.219
C01167=1058.408,-57.523,434.150,171.178,27.822,155.219
C01168=1058.401,-57.772,434.161,171.176,27.820,155.219
C01169=1058.395,-58.022,434.174,171.174,27.818,155.218
C01170=1058.389,-58.272,434.185,171.173,27.816,155.218
C01171=1058.382,-58.522,434.197,171.171,27.815,155.218
C01172=1058.377,-58.771,434.209,171.169,27.813,155.218
C01173=1058.370,-59.021,434.221,171.168,27.811,155.218
C01174=1058.364,-59.271,434.234,171.166,27.810,155.218
C01175=1058.358,-59.520,434.246,171.164,27.808,155.218
C01176=1058.352,-59.770,434.257,171.162,27.806,155.217
C01177=1058.346,-60.019,434.269,171.161,27.805,155.217
C01178=1058.339,-60.269,434.281,171.159,27.804,155.217
C01179=1058.333,-60.519,434.293,171.157,27.802,155.217
C01180=1058.327,-60.768,434.305,171.155,27.800,155.217
C01181=1058.321,-61.018,434.317,171.154,27.799,155.217
C01182=1058.314,-61.268,434.329,171.152,27.797,155.217
C01183=1058.308,-61.517,434.341,171.150,27.795,155.216
C01184=1058.302,-61.766,434.353,171.149,27.794,155.216
C01185=1058.296,-62.016,434.364,171.147,27.792,155.216
C01186=1058.289,-62.266,434.376,171.145,27.790,155.216
C01187=1058.283,-62.516,434.389,171.143,27.789,155.216
C01188=1058.278,-62.765,434.399,171.142,27.787,155.216
C01189=1058.271,-63.015,434.411,171.140,27.785,155.216
C01190=1058.265,-63.265,434.424,171.137,27.784,155.216
C01191=1058.259,-63.514,434.435,171.136,27.782,155.215
C01192=1058.253,-63.764,434.447,171.134,27.781,155.215
C01193=1058.247,-64.014,434.459,171.132,27.779,155.215
C01194=1058.241,-64.263,434.470,171.130,27.777,155.215
C01195=1058.234,-64.513,434.482,171.129,27.775,155.215
C01196=1058.229,-64.763,434.495,171.127,27.774,155.215
C01197=1058.223,-65.012,434.506,171.125,27.772,155.215
C01198=1058.216,-65.262,434.518,171.123,27.771,155.215
C01199=1058.210,-65.511,434.530,171.122,27.769,155.214
C01200=1058.205,-65.761,434.541,171.120,27.768,155.214
C01201=1058.198,-66.011,434.553,171.118,27.766,155.214
C01202=1058.191,-66.292,434.566,171.117,27.764,155.214
C01203=1058.185,-66.572,434.579,171.114,27.762,155.214
C01204=1058.177,-66.853,434.592,171.112,27.761,155.214
C01205=1058.171,-67.134,434.605,171.111,27.759,155.214
C01206=1058.165,-67.383,434.617,171.109,27.757,155.213
C01207=1058.159,-67.633,434.628,171.107,27.756,155.213
C01208=1058.152,-67.883,434.640,171.105,27.754,155.213
C01209=1058.147,-68.132,434.652,171.104,27.752,155.213
C01210=1058.140,-68.382,434.664,171.101,27.751,155.213
C01211=1058.134,-68.631,434.675,171.099,27.749,155.213
C01212=1058.128,-68.881,434.687,171.098,27.748,155.213
C01213=1058.122,-69.131,434.699,171.096,27.746,155.213
C01214=1058.116,-69.381,434.710,171.094,27.744,155.212
C01215=1058.110,-69.630,434.722,171.092,27.743,155.212
C01216=1058.104,-69.880,434.733,171.091,27.741,155.212
C01217=1058.098,-70.130,434.745,171.089,27.740,155.212
C01218=1058.092,-70.379,434.756,171.087,27.738,155.212
C01219=1058.086,-70.629,434.768,171.085,27.736,155.212
C01220=1058.080,-70.878,434.779,171.084,27.735,155.212
C01221=1058.073,-71.128,434.790,171.082,27.734,155.212
C01222=1058.068,-71.377,434.803,171.080,27.732,155.212
C01223=1058.062,-71.628,434.814,171.079,27.730,155.211
C01224=1058.055,-71.877,434.826,171.077,27.729,155.211
C01225=1058.049,-72.127,434.837,171.075,27.728,155.211
C01226=1058.043,-72.377,434.849,171.073,27.726,155.211
C01227=1058.038,-72.626,434.860,171.072,27.724,155.211
C01228=1058.031,-72.876,434.871,171.069,27.723,155.211
C01229=1058.025,-73.125,434.883,171.067,27.721,155.211
C01230=1058.019,-73.375,434.894,171.065,27.719,155.211
C01231=1058.014,-73.625,434.906,171.064,27.718,155.211
C01232=1058.007,-73.875,434.918,171.062,27.717,155.210
C01233=1058.002,-74.124,434.928,171.060,27.715,155.210
C01234=1057.995,-74.374,434.940,171.058,27.714,155.210
C01235=1057.989,-74.623,434.951,171.057,27.712,155.210
C01236=1057.983,-74.873,434.963,171.055,27.711,155.210
C01237=1057.977,-75.123,434.973,171.053,27.709,155.210
C01238=1057.971,-75.373,434.985,171.052,27.708,155.210
C01239=1057.965,-75.622,434.996,171.050,27.707,155.210
C01240=1057.958,-75.872,435.007,171.048,27.705,155.210
C01241=1057.952,-76.121,435.019,171.046,27.704,155.210
C01242=1057.946,-76.371,435.030,171.044,27.702,155.210
C01243=1057.940,-76.621,435.041,171.042,27.701,155.210
C01244=1057.934,-76.871,435.052,171.040,27.699,155.209
C01245=1057.928,-77.120,435.064,171.038,27.698,155.209
C01246=1057.921,-77.370,435.075,171.037,27.696,155.209
C01247=1057.915,-77.619,435.086,171.035,27.695,155.209
C01248=1057.909,-77.869,435.097,171.033,27.694,155.209
C01249=1057.903,-78.118,435.108,171.031,27.693,155.209
C01250=1057.896,-78.368,435.120,171.029,27.691,155.209
C01251=1057.891,-78.618,435.130,171.028,27.690,155.209
C01252=1057.884,-78.868,435.142,171.026,27.688,155.209
C01253=1057.879,-79.118,435.153,171.024,27.687,155.209
C01254=1057.872,-79.367,435.165,171.022,27.685,155.209
C01255=1057.866,-79.617,435.175,171.021,27.684,155.208
C01256=1057.860,-79.866,435.186,171.018,27.682,155.208
C01257=1057.854,-80.116,435.198,171.016,27.681,155.208
C01258=1057.848,-80.366,435.208,171.014,27.680,155.208
C01259=1057.841,-80.616,435.219,171.013,27.679,155.208
C01260=1057.836,-80.865,435.230,171.011,27.677,155.208
C01261=1057.829,-81.115,435.241,171.009,27.676,155.208
C01262=1057.822,-81.364,435.252,171.007,27.675,155.208
C01263=1057.816,-81.614,435.263,171.006,27.673,155.208
C01264=1057.810,-81.864,435.274,171.004,27.672,155.208
C01265=1057.803,-82.114,435.285,171.002,27.671,155.208
C01266=1057.797,-82.397,435.297,170.999,27.669,155.208
C01267=1057.789,-82.679,435.310,170.998,27.668,155.208
C01268=1057.783,-82.962,435.322,170.996,27.667,155.208
C01269=1057.775,-83.245,435.334,170.993,27.665,155.208
C01270=1057.769,-83.495,435.346,170.991,27.664,155.208
C01271=1057.763,-83.745,435.356,170.990,27.662,155.207
C01272=1057.756,-83.994,435.367,170.988,27.661,155.207
C01273=1057.751,-84.244,435.378,170.986,27.660,155.207
C01274=1057.745,-84.493,435.389,170.984,27.659,155.207
C01275=1057.738,-84.744,435.400,170.982,27.657,155.207
C01276=1057.732,-84.993,435.410,170.981,27.656,155.207
C01277=1057.726,-85.243,435.422,170.979,27.655,155.207
C01278=1057.720,-85.492,435.433,170.976,27.654,155.207
C01279=1057.713,-85.742,435.443,170.974,27.653,155.207
C01280=1057.707,-85.992,435.454,170.973,27.651,155.207
C01281=1057.701,-86.241,435.465,170.971,27.650,155.207
C01282=1057.694,-86.491,435.476,170.969,27.649,155.207
C01283=1057.689,-86.741,435.486,170.967,27.648,155.207
C01284=1057.683,-86.991,435.497,170.965,27.647,155.207
C01285=1057.676,-87.241,435.507,170.964,27.645,155.207
C01286=1057.670,-87.490,435.518,170.962,27.644,155.207
C01287=1057.665,-87.740,435.529,170.960,27.643,155.207
C01288=1057.657,-87.990,435.540,170.958,27.642,155.207
C01289=1057.652,-88.239,435.551,170.956,27.640,155.207
C01290=1057.646,-88.488,435.561,170.954,27.639,155.207
C01291=1057.639,-88.738,435.572,170.952,27.638,155.207
C01292=1057.633,-88.988,435.583,170.950,27.637,155.207
C01293=1057.628,-89.238,435.593,170.948,27.636,155.207
C01294=1057.621,-89.488,435.604,170.947,27.634,155.207
C01295=1057.615,-89.737,435.615,170.945,27.633,155.206
C01296=1057.609,-89.987,435.626,170.943,27.632,155.206
C01297=1057.603,-90.236,435.636,170.941,27.631,155.206
C01298=1057.596,-90.486,435.647,170.940,27.629,155.206
C01299=1057.591,-90.736,435.657,170.938,27.628,155.206
C01300=1057.584,-90.985,435.667,170.935,27.627,155.206
C01301=1057.578,-91.236,435.679,170.933,27.626,155.206
C01302=1057.572,-91.485,435.689,170.931,27.625,155.206
C01303=1057.566,-91.734,435.700,170.930,27.624,155.206
C01304=1057.560,-91.984,435.710,170.928,27.623,155.206
C01305=1057.553,-92.234,435.721,170.926,27.622,155.206
C01306=1057.548,-92.484,435.732,170.924,27.620,155.206
C01307=1057.542,-92.733,435.742,170.923,27.619,155.206
C01308=1057.536,-92.983,435.752,170.921,27.618,155.206
C01309=1057.529,-93.233,435.763,170.919,27.617,155.206
C01310=1057.523,-93.482,435.774,170.917,27.615,155.206
C01311=1057.517,-93.732,435.784,170.914,27.614,155.206
C01312=1057.512,-93.982,435.795,170.913,27.613,155.206
C01313=1057.505,-94.232,435.805,170.911,27.612,155.206
C01314=1057.499,-94.481,435.816,170.909,27.611,155.206
C01315=1057.493,-94.731,435.826,170.907,27.610,155.206
C01316=1057.487,-94.981,435.837,170.905,27.609,155.206
C01317=1057.481,-95.230,435.847,170.904,27.608,155.206
C01318=1057.474,-95.481,435.857,170.902,27.606,155.206
C01319=1057.469,-95.730,435.868,170.900,27.605,155.206
C01320=1057.462,-95.979,435.879,170.898,27.604,155.206
C01321=1057.457,-96.230,435.889,170.896,27.603,155.206
C01322=1057.450,-96.479,435.899,170.894,27.602,155.206
C01323=1057.445,-96.728,435.910,170.892,27.601,155.206
C01324=1057.439,-96.979,435.920,170.890,27.600,155.206
C01325=1057.432,-97.228,435.931,170.888,27.599,155.206
C01326=1057.427,-97.478,435.941,170.886,27.597,155.206
C01327=1057.420,-97.727,435.951,170.885,27.596,155.206
C01328=1057.414,-97.977,435.961,170.883,27.595,155.206
C01329=1057.408,-98.227,435.972,170.881,27.595,155.206
C01330=1057.401,-98.512,435.984,170.878,27.593,155.206
C01331=1057.393,-98.798,435.995,170.876,27.592,155.206
C01332=1057.386,-99.082,436.007,170.875,27.591,155.206
C01333=1057.379,-99.368,436.018,170.872,27.590,155.206
C01334=1057.373,-99.618,436.029,170.870,27.589,155.206
C01335=1057.367,-99.867,436.040,170.868,27.588,155.206
C01336=1057.361,-100.117,436.049,170.866,27.587,155.206
C01337=1057.355,-100.366,436.059,170.865,27.586,155.206
C01338=1057.349,-100.616,436.070,170.863,27.585,155.206
C01339=1057.342,-100.866,436.080,170.861,27.584,155.206
C01340=1057.336,-101.116,436.090,170.858,27.583,155.206
C01341=1057.330,-101.366,436.100,170.856,27.582,155.206
C01342=1057.324,-101.615,436.110,170.855,27.581,155.206
C01343=1057.318,-101.865,436.120,170.853,27.580,155.206
C01344=1057.312,-102.114,436.131,170.851,27.579,155.206
C01345=1057.306,-102.364,436.140,170.849,27.578,155.206
C01346=1057.299,-102.614,436.151,170.847,27.577,155.206
C01347=1057.293,-102.864,436.161,170.845,27.576,155.206
C01348=1057.287,-103.113,436.171,170.844,27.575,155.206
C01349=1057.281,-103.363,436.181,170.841,27.574,155.206
C01350=1057.275,-103.613,436.191,170.839,27.573,155.206
C01351=1057.269,-103.862,436.201,170.837,27.572,155.206
C01352=1057.263,-104.112,436.211,170.835,27.572,155.206
C01353=1057.257,-104.362,436.222,170.834,27.570,155.206
C01354=1057.251,-104.612,436.231,170.832,27.569,155.206
C01355=1057.245,-104.861,436.241,170.830,27.569,155.206
C01356=1057.238,-105.111,436.252,170.828,27.568,155.206
C01357=1057.232,-105.361,436.262,170.826,27.567,155.206
C01358=1057.226,-105.611,436.271,170.824,27.566,155.206
C01359=1057.219,-105.860,436.282,170.822,27.565,155.206
C01360=1057.213,-106.110,436.291,170.820,27.564,155.206
C01361=1057.208,-106.360,436.301,170.818,27.563,155.206
C01362=1057.201,-106.609,436.312,170.816,27.562,155.206
C01363=1057.195,-106.859,436.321,170.814,27.561,155.206
C01364=1057.189,-107.109,436.331,170.812,27.561,155.206
C01365=1057.184,-107.359,436.341,170.811,27.559,155.206
C01366=1057.177,-107.608,436.351,170.809,27.559,155.206
C01367=1057.171,-107.858,436.361,170.807,27.558,155.206
C01368=1057.165,-108.108,436.370,170.804,27.557,155.206
C01369=1057.159,-108.358,436.380,170.802,27.556,155.206
C01370=1057.152,-108.607,436.390,170.800,27.556,155.206
C01371=1057.147,-108.857,436.400,170.799,27.554,155.206
C01372=1057.140,-109.107,436.410,170.797,27.554,155.206
C01373=1057.134,-109.357,436.420,170.795,27.553,155.206
C01374=1057.127,-109.606,436.430,170.793,27.552,155.206
C01375=1057.121,-109.856,436.440,170.791,27.551,155.206
C01376=1057.115,-110.106,436.449,170.789,27.551,155.206
C01377=1057.109,-110.356,436.459,170.787,27.549,155.206
C01378=1057.103,-110.606,436.468,170.785,27.549,155.207
C01379=1057.096,-110.855,436.479,170.783,27.548,155.207
C01380=1057.091,-111.105,436.489,170.781,27.547,155.207
C01381=1057.084,-111.355,436.498,170.779,27.546,155.207
C01382=1057.078,-111.604,436.508,170.777,27.546,155.207
C01383=1057.072,-111.854,436.517,170.775,27.545,155.207
C01384=1057.066,-112.104,436.527,170.774,27.544,155.207
C01385=1057.060,-112.354,436.537,170.772,27.544,155.207
C01386=1057.053,-112.603,436.547,170.769,27.542,155.207
C01387=1057.047,-112.853,436.556,170.767,27.542,155.207
C01388=1057.042,-113.102,436.566,170.765,27.541,155.207
C01389=1057.035,-113.352,436.575,170.763,27.540,155.207
C01390=1057.029,-113.602,436.585,170.762,27.540,155.207
C01391=1057.023,-113.851,436.594,170.760,27.539,155.207
C01392=1057.018,-114.101,436.605,170.758,27.538,155.207
C01393=1057.011,-114.351,436.614,170.756,27.538,155.207
C01394=1057.004,-114.635,436.624,170.753,27.536,155.207
C01395=1056.997,-114.918,436.635,170.751,27.536,155.207
C01396=1056.990,-115.202,436.647,170.748,27.535,155.208
C01397=1056.983,-115.486,436.658,170.747,27.534,155.208
C01398=1056.976,-115.736,436.667,170.745,27.533,155.208
C01399=1056.970,-115.986,436.677,170.743,27.533,155.208
C01400=1056.965,-116.235,436.686,170.741,27.532,155.208
C01401=1056.959,-116.485,436.696,170.739,27.531,155.208
C01402=1056.952,-116.734,436.705,170.737,27.531,155.208
C01403=1056.946,-116.984,436.715,170.734,27.530,155.208
C01404=1056.940,-117.234,436.724,170.733,27.529,155.208
C01405=1056.934,-117.484,436.734,170.731,27.528,155.208
C01406=1056.928,-117.734,436.743,170.729,27.528,155.208
C01407=1056.922,-117.983,436.753,170.727,27.527,155.208
C01408=1056.915,-118.233,436.763,170.725,27.526,155.208
C01409=1056.908,-118.483,436.772,170.723,27.526,155.208
C01410=1056.902,-118.732,436.781,170.721,27.525,155.208
C01411=1056.897,-118.982,436.790,170.720,27.525,155.209
C01412=1056.891,-119.232,436.799,170.717,27.524,155.209
C01413=1056.885,-119.482,436.809,170.715,27.524,155.209
C01414=1056.878,-119.732,436.818,170.713,27.523,155.209
C01415=1056.872,-119.981,436.828,170.711,27.522,155.209
C01416=1056.866,-120.231,436.837,170.709,27.522,155.209
C01417=1056.860,-120.481,436.847,170.707,27.521,155.209
C01418=1056.854,-120.731,436.857,170.705,27.521,155.209
C01419=1056.847,-120.980,436.865,170.704,27.520,155.209
C01420=1056.842,-121.230,436.874,170.701,27.519,155.209
C01421=1056.835,-121.480,436.884,170.699,27.518,155.209
C01422=1056.829,-121.730,436.893,170.697,27.518,155.209
C01423=1056.823,-121.979,436.903,170.695,27.517,155.209
C01424=1056.817,-122.229,436.912,170.693,27.517,155.210
C01425=1056.812,-122.479,436.921,170.691,27.516,155.210
C01426=1056.805,-122.728,436.930,170.689,27.516,155.210
C01427=1056.799,-122.978,436.939,170.688,27.515,155.210
C01428=1056.792,-123.228,436.949,170.686,27.515,155.210
C01429=1056.786,-123.478,436.958,170.683,27.514,155.210
C01430=1056.780,-123.728,436.967,170.681,27.513,155.210
C01431=1056.775,-123.977,436.977,170.679,27.513,155.210
C01432=1056.768,-124.227,436.986,170.677,27.512,155.210
C01433=1056.762,-124.477,436.995,170.675,27.512,155.210
C01434=1056.756,-124.727,437.004,170.673,27.511,155.211
C01435=1056.750,-124.977,437.014,170.671,27.511,155.211
C01436=1056.743,-125.226,437.022,170.670,27.510,155.211
C01437=1056.737,-125.475,437.032,170.668,27.510,155.211
C01438=1056.731,-125.726,437.041,170.665,27.509,155.211
C01439=1056.725,-125.976,437.050,170.663,27.509,155.211
C01440=1056.718,-126.225,437.059,170.661,27.508,155.211
C01441=1056.713,-126.475,437.068,170.659,27.508,155.211
C01442=1056.707,-126.725,437.077,170.657,27.507,155.211
C01443=1056.700,-126.974,437.086,170.655,27.507,155.211
C01444=1056.694,-127.224,437.095,170.653,27.506,155.211
C01445=1056.688,-127.474,437.105,170.652,27.506,155.212
C01446=1056.682,-127.723,437.114,170.650,27.505,155.212
C01447=1056.676,-127.974,437.123,170.647,27.505,155.212
C01448=1056.672,-128.223,437.132,170.645,27.503,155.212
C01449=1056.668,-128.473,437.143,170.643,27.502,155.212
C01450=1056.667,-128.725,437.155,170.643,27.500,155.211
C01451=1056.666,-128.975,437.167,170.641,27.497,155.211
C01452=1056.667,-129.225,437.180,170.640,27.493,155.211
C01453=1056.668,-129.475,437.193,170.638,27.489,155.210
C01454=1056.673,-129.727,437.207,170.638,27.485,155.209
C01455=1056.676,-129.978,437.222,170.637,27.479,155.208
C01456=1056.682,-130.229,437.238,170.637,27.474,155.207
C01457=1056.689,-130.478,437.253,170.636,27.468,155.206
C01458=1056.315,-130.501,437.048,170.589,27.632,155.240
C01459=1056.308,-130.252,437.032,170.589,27.638,155.241
C01460=1056.303,-130.001,437.017,170.590,27.644,155.242
C01461=1056.297,-129.750,437.002,170.590,27.649,155.242
C01462=1056.295,-129.498,436.987,170.591,27.654,155.243
C01463=1056.294,-129.248,436.974,170.592,27.657,155.244
C01464=1056.293,-128.998,436.961,170.593,27.661,155.244
C01465=1056.293,-128.747,436.950,170.595,27.664,155.245
C01466=1056.295,-128.497,436.938,170.596,27.666,155.245
C01467=1056.298,-128.246,436.927,170.598,27.668,155.245
C01468=1056.302,-127.996,436.917,170.600,27.670,155.245
C01469=1056.308,-127.747,436.908,170.602,27.670,155.245
C01470=1056.313,-127.497,436.899,170.604,27.671,155.245
C01471=1056.320,-127.247,436.889,170.605,27.671,155.245
C01472=1056.326,-126.998,436.880,170.607,27.672,155.245
C01473=1056.332,-126.748,436.872,170.609,27.672,155.245
C01474=1056.338,-126.498,436.862,170.611,27.673,155.245
C01475=1056.344,-126.248,436.853,170.613,27.672,155.244
C01476=1056.351,-125.998,436.845,170.616,27.673,155.244
C01477=1056.357,-125.748,436.835,170.618,27.674,155.244
C01478=1056.362,-125.499,436.826,170.620,27.674,155.244
C01479=1056.369,-125.249,436.816,170.622,27.675,155.244
C01480=1056.375,-124.999,436.808,170.624,27.675,155.244
C01481=1056.381,-124.750,436.798,170.625,27.676,155.244
C01482=1056.388,-124.500,436.789,170.627,27.676,155.244
C01483=1056.394,-124.250,436.781,170.629,27.677,155.244
C01484=1056.400,-124.001,436.771,170.632,27.677,155.243
C01485=1056.406,-123.751,436.762,170.634,27.678,155.243
C01486=1056.412,-123.501,436.752,170.636,27.678,155.243
C01487=1056.418,-123.251,436.743,170.638,27.679,155.243
C01488=1056.424,-123.001,436.734,170.640,27.679,155.243
C01489=1056.430,-122.752,436.725,170.642,27.680,155.243
C01490=1056.437,-122.502,436.716,170.643,27.680,155.243
C01491=1056.443,-122.252,436.706,170.645,27.681,155.243
C01492=1056.449,-122.003,436.696,170.647,27.682,155.243
C01493=1056.455,-121.752,436.688,170.650,27.683,155.243
C01494=1056.461,-121.502,436.678,170.652,27.683,155.243
C01495=1056.467,-121.253,436.669,170.654,27.684,155.243
C01496=1056.473,-121.004,436.660,170.656,27.684,155.242
C01497=1056.480,-120.754,436.650,170.658,27.684,155.242
C01498=1056.486,-120.504,436.641,170.660,27.685,155.242
C01499=1056.492,-120.254,436.632,170.661,27.685,155.242
C01500=1056.498,-120.004,436.622,170.663,27.686,155.242
C01501=1056.504,-119.754,436.613,170.666,27.687,155.242
C01502=1056.510,-119.505,436.604,170.668,27.688,155.242
C01503=1056.516,-119.255,436.594,170.670,27.688,155.242
C01504=1056.522,-119.005,436.584,170.672,27.689,155.242
C01505=1056.528,-118.756,436.575,170.674,27.689,155.242
C01506=1056.535,-118.506,436.566,170.676,27.690,155.242
C01507=1056.541,-118.256,436.556,170.677,27.691,155.242
C01508=1056.547,-118.007,436.547,170.679,27.691,155.242
C01509=1056.554,-117.757,436.537,170.681,27.692,155.241
C01510=1056.560,-117.507,436.528,170.684,27.693,155.241
C01511=1056.565,-117.258,436.518,170.686,27.693,155.241
C01512=1056.571,-117.007,436.510,170.688,27.694,155.241
C01513=1056.577,-116.758,436.500,170.690,27.695,155.241
C01514=1056.583,-116.508,436.490,170.691,27.695,155.241
C01515=1056.590,-116.258,436.481,170.693,27.696,155.241
C01516=1056.596,-116.008,436.471,170.695,27.697,155.241
C01517=1056.602,-115.758,436.462,170.697,27.697,155.241
C01518=1056.608,-115.509,436.452,170.700,27.698,155.241
C01519=1056.615,-115.225,436.441,170.702,27.699,155.241
C01520=1056.622,-114.941,436.430,170.704,27.699,155.241
C01521=1056.630,-114.658,436.420,170.706,27.700,155.241
C01522=1056.637,-114.374,436.408,170.708,27.701,155.241
C01523=1056.643,-114.124,436.399,170.710,27.702,155.240
C01524=1056.649,-113.875,436.390,170.712,27.702,155.240
C01525=1056.654,-113.625,436.380,170.715,27.704,155.240
C01526=1056.660,-113.375,436.370,170.717,27.704,155.240
C01527=1056.666,-113.125,436.360,170.719,27.705,155.240
C01528=1056.673,-112.875,436.351,170.720,27.706,155.240
C01529=1056.679,-112.626,436.341,170.722,27.706,155.240
C01530=1056.685,-112.376,436.331,170.724,27.707,155.240
C01531=1056.691,-112.127,436.321,170.726,27.708,155.240
C01532=1056.698,-111.877,436.312,170.728,27.708,155.240
C01533=1056.704,-111.627,436.302,170.730,27.709,155.240
C01534=1056.710,-111.377,436.293,170.733,27.710,155.240
C01535=1056.716,-111.127,436.283,170.734,27.711,155.240
C01536=1056.722,-110.878,436.272,170.736,27.712,155.240
C01537=1056.728,-110.628,436.263,170.738,27.713,155.240
C01538=1056.734,-110.378,436.253,170.740,27.713,155.240
C01539=1056.740,-110.129,436.244,170.742,27.714,155.240
C01540=1056.747,-109.879,436.234,170.744,27.715,155.240
C01541=1056.753,-109.630,436.224,170.746,27.715,155.240
C01542=1056.759,-109.380,436.214,170.748,27.717,155.240
C01543=1056.765,-109.130,436.205,170.750,27.717,155.239
C01544=1056.772,-108.880,436.195,170.752,27.718,155.239
C01545=1056.777,-108.630,436.185,170.754,27.719,155.239
C01546=1056.784,-108.381,436.175,170.756,27.720,155.239
C01547=1056.790,-108.130,436.165,170.758,27.720,155.239
C01548=1056.796,-107.881,436.155,170.759,27.721,155.239
C01549=1056.803,-107.631,436.146,170.761,27.722,155.239
C01550=1056.809,-107.382,436.135,170.763,27.723,155.239
C01551=1056.815,-107.131,436.125,170.766,27.724,155.239
C01552=1056.821,-106.882,436.116,170.768,27.725,155.239
C01553=1056.827,-106.633,436.105,170.769,27.726,155.239
C01554=1056.833,-106.383,436.096,170.771,27.726,155.239
C01555=1056.840,-106.133,436.086,170.773,27.727,155.239
C01556=1056.845,-105.883,436.076,170.775,27.728,155.239
C01557=1056.851,-105.634,436.066,170.777,27.729,155.239
C01558=1056.858,-105.384,436.056,170.779,27.730,155.239
C01559=1056.866,-105.028,436.041,170.781,27.731,155.239
C01560=1056.875,-104.672,436.027,170.784,27.733,155.239
C01561=1056.884,-104.317,436.013,170.787,27.733,155.239
C01562=1056.892,-103.961,435.998,170.790,27.735,155.239
C01563=1056.899,-103.711,435.989,170.792,27.736,155.239
C01564=1056.905,-103.462,435.978,170.794,27.737,155.239
C01565=1056.910,-103.212,435.968,170.796,27.738,155.239
C01566=1056.917,-102.962,435.959,170.798,27.739,155.239
C01567=1056.924,-102.712,435.948,170.800,27.740,155.239
C01568=1056.929,-102.462,435.938,170.802,27.741,155.239
C01569=1056.936,-102.213,435.928,170.804,27.741,155.239
C01570=1056.942,-101.963,435.918,170.805,27.743,155.239
C01571=1056.948,-101.713,435.907,170.807,27.744,155.239
C01572=1056.954,-101.464,435.898,170.809,27.745,155.239
C01573=1056.960,-101.214,435.887,170.812,27.745,155.239
C01574=1056.966,-100.964,435.877,170.814,27.747,155.239
C01575=1056.972,-100.714,435.867,170.815,27.748,155.239
C01576=1056.979,-100.465,435.857,170.817,27.749,155.239
C01577=1056.984,-100.214,435.847,170.819,27.749,155.239
C01578=1056.991,-99.965,435.837,170.821,27.750,155.239
C01579=1056.996,-99.751,435.828,170.823,27.751,155.239
C01580=1057.001,-99.537,435.819,170.825,27.752,155.239
C01581=1057.007,-99.322,435.810,170.826,27.753,155.239
C01582=1057.012,-99.107,435.802,170.827,27.754,155.239
C01583=1057.017,-98.893,435.793,170.829,27.755,155.239
C01584=1057.023,-98.679,435.784,170.831,27.755,155.239
C01585=1057.028,-98.464,435.776,170.833,27.756,155.239
C01586=1057.033,-98.250,435.766,170.835,27.758,155.239
C01587=1057.039,-97.999,435.756,170.836,27.758,155.239
C01588=1057.046,-97.750,435.746,170.838,27.759,155.239
C01589=1057.052,-97.501,435.735,170.840,27.760,155.239
C01590=1057.058,-97.251,435.725,170.842,27.761,155.239
C01591=1057.064,-97.002,435.715,170.844,27.762,155.239
C01592=1057.070,-96.751,435.704,170.846,27.763,155.239
C01593=1057.076,-96.501,435.693,170.847,27.765,155.239
C01594=1057.082,-96.252,435.683,170.849,27.766,155.239
C01595=1057.088,-96.002,435.673,170.852,27.767,155.239
C01596=1057.094,-95.753,435.663,170.854,27.768,155.239
C01597=1057.101,-95.503,435.651,170.855,27.769,155.239
C01598=1057.107,-95.253,435.642,170.857,27.770,155.239
C01599=1057.113,-95.003,435.631,170.859,27.771,155.239
C01600=1057.118,-94.754,435.620,170.861,27.772,155.239
C01601=1057.124,-94.504,435.611,170.863,27.773,155.239
C01602=1057.131,-94.254,435.599,170.864,27.775,155.239
C01603=1057.137,-94.005,435.589,170.866,27.776,155.239
C01604=1057.143,-93.755,435.579,170.868,27.777,155.239
C01605=1057.148,-93.505,435.568,170.870,27.778,155.239
C01606=1057.155,-93.256,435.558,170.873,27.779,155.239
C01607=1057.161,-93.006,435.546,170.874,27.780,155.239
C01608=1057.167,-92.756,435.537,170.876,27.781,155.239
C01609=1057.173,-92.506,435.526,170.878,27.782,155.239
C01610=1057.179,-92.257,435.515,170.880,27.783,155.239
C01611=1057.186,-92.007,435.504,170.882,27.785,155.239
C01612=1057.191,-91.757,435.494,170.883,27.786,155.239
C01613=1057.197,-91.507,435.483,170.885,27.787,155.239
C01614=1057.204,-91.258,435.473,170.887,27.788,155.239
C01615=1057.210,-91.008,435.462,170.889,27.789,155.239
C01616=1057.216,-90.759,435.452,170.892,27.791,155.239
C01617=1057.222,-90.509,435.441,170.893,27.792,155.239
C01618=1057.228,-90.259,435.430,170.895,27.793,155.240
C01619=1057.235,-90.009,435.420,170.897,27.794,155.240
C01620=1057.240,-89.760,435.409,170.899,27.795,155.240
C01621=1057.246,-89.510,435.398,170.901,27.796,155.240
C01622=1057.253,-89.261,435.388,170.902,27.798,155.240
C01623=1057.259,-89.010,435.377,170.904,27.799,155.240
C01624=1057.264,-88.761,435.366,170.906,27.800,155.240
C01625=1057.272,-88.511,435.356,170.908,27.801,155.240
C01626=1057.277,-88.262,435.345,170.910,27.802,155.240
C01627=1057.283,-88.012,435.334,170.912,27.804,155.240
C01628=1057.290,-87.762,435.323,170.914,27.805,155.240
C01629=1057.296,-87.513,435.313,170.916,27.806,155.240
C01630=1057.302,-87.263,435.302,170.918,27.807,155.240
C01631=1057.309,-87.013,435.291,170.919,27.809,155.240
C01632=1057.314,-86.764,435.280,170.921,27.810,155.240
C01633=1057.320,-86.513,435.270,170.923,27.811,155.240
C01634=1057.327,-86.264,435.259,170.925,27.812,155.240
C01635=1057.333,-86.014,435.248,170.927,27.813,155.240
C01636=1057.339,-85.764,435.237,170.928,27.815,155.240
C01637=1057.345,-85.515,435.227,170.931,27.816,155.240
C01638=1057.351,-85.265,435.216,170.933,27.817,155.240
C01639=1057.358,-85.015,435.205,170.935,27.819,155.240
C01640=1057.364,-84.766,435.195,170.936,27.820,155.240
C01641=1057.370,-84.516,435.183,170.938,27.821,155.241
C01642=1057.376,-84.266,435.172,170.940,27.822,155.241
C01643=1057.382,-84.016,435.161,170.942,27.823,155.241
C01644=1057.389,-83.767,435.151,170.944,27.825,155.241
C01645=1057.395,-83.518,435.140,170.945,27.826,155.241
C01646=1057.401,-83.267,435.129,170.947,27.827,155.241
C01647=1057.408,-82.985,435.116,170.950,27.829,155.241
C01648=1057.415,-82.702,435.104,170.952,27.830,155.241
C01649=1057.422,-82.419,435.092,170.953,27.831,155.241
C01650=1057.429,-82.135,435.079,170.956,27.833,155.241
C01651=1057.436,-81.886,435.069,170.958,27.834,155.241
C01652=1057.442,-81.636,435.057,170.960,27.835,155.241
C01653=1057.448,-81.386,435.047,170.961,27.837,155.241
C01654=1057.454,-81.138,435.035,170.963,27.838,155.241
C01655=1057.461,-80.888,435.024,170.965,27.839,155.241
C01656=1057.467,-80.638,435.013,170.967,27.841,155.241
C01657=1057.473,-80.388,435.002,170.969,27.842,155.241
C01658=1057.479,-80.139,434.991,170.971,27.843,155.241
C01659=1057.486,-79.889,434.981,170.973,27.845,155.242
C01660=1057.492,-79.639,434.970,170.975,27.846,155.242
C01661=1057.498,-79.389,434.959,170.977,27.847,155.242
C01662=1057.504,-79.140,434.947,170.978,27.848,155.242
C01663=1057.510,-78.890,434.936,170.980,27.850,155.242
C01664=1057.516,-78.640,434.925,170.982,27.851,155.242
C01665=1057.523,-78.390,434.914,170.984,27.852,155.242
C01666=1057.528,-78.141,434.903,170.985,27.854,155.242
C01667=1057.535,-77.891,434.891,170.987,27.855,155.242
C01668=1057.541,-77.642,434.880,170.989,27.857,155.242
C01669=1057.547,-77.392,434.869,170.991,27.858,155.242
C01670=1057.553,-77.142,434.858,170.992,27.860,155.242
C01671=1057.559,-76.892,434.846,170.995,27.861,155.242
C01672=1057.565,-76.643,434.835,170.997,27.863,155.243
C01673=1057.571,-76.393,434.824,170.999,27.864,155.243
C01674=1057.578,-76.144,434.813,171.000,27.865,155.243
C01675=1057.585,-75.894,434.801,171.002,27.866,155.243
C01676=1057.590,-75.645,434.791,171.004,27.868,155.243
C01677=1057.597,-75.394,434.779,171.006,27.869,155.243
C01678=1057.603,-75.145,434.768,171.008,27.871,155.243
C01679=1057.609,-74.895,434.757,171.009,27.872,155.243
C01680=1057.615,-74.646,434.746,171.011,27.874,155.243
C01681=1057.621,-74.396,434.734,171.013,27.875,155.243
C01682=1057.627,-74.147,434.723,171.015,27.876,155.243
C01683=1057.634,-73.897,434.712,171.016,27.878,155.244
C01684=1057.639,-73.647,434.699,171.018,27.879,155.244
C01685=1057.645,-73.397,434.688,171.021,27.881,155.244
C01686=1057.651,-73.148,434.677,171.022,27.883,155.244
C01687=1057.658,-72.898,434.665,171.024,27.884,155.244
C01688=1057.663,-72.649,434.654,171.026,27.885,155.244
C01689=1057.669,-72.398,434.643,171.028,27.887,155.244
C01690=1057.675,-72.149,434.631,171.029,27.889,155.244
C01691=1057.681,-71.899,434.620,171.031,27.890,155.244
C01692=1057.687,-71.650,434.608,171.033,27.892,155.245
C01693=1057.694,-71.400,434.597,171.035,27.893,155.245
C01694=1057.699,-71.151,434.585,171.036,27.895,155.245
C01695=1057.705,-70.901,434.573,171.038,27.896,155.245
C01696=1057.712,-70.651,434.562,171.040,27.898,155.245
C01697=1057.718,-70.402,434.551,171.042,27.899,155.245
C01698=1057.723,-70.151,434.539,171.043,27.901,155.245
C01699=1057.729,-69.902,434.527,171.045,27.902,155.245
C01700=1057.736,-69.652,434.516,171.047,27.904,155.245
C01701=1057.742,-69.403,434.504,171.049,27.905,155.246
C01702=1057.747,-69.153,434.493,171.051,27.907,155.246
C01703=1057.753,-68.904,434.481,171.053,27.908,155.246
C01704=1057.760,-68.654,434.470,171.055,27.910,155.246
C01705=1057.766,-68.404,434.458,171.057,27.912,155.246
C01706=1057.772,-68.155,434.446,171.058,27.913,155.246
C01707=1057.778,-67.905,434.434,171.060,27.915,155.246
C01708=1057.784,-67.656,434.423,171.062,27.916,155.246
C01709=1057.790,-67.406,434.411,171.063,27.918,155.246
C01710=1057.796,-67.156,434.399,171.065,27.920,155.247
C01711=1057.803,-66.875,434.387,171.067,27.921,155.247
C01712=1057.810,-66.594,434.374,171.070,27.923,155.247
C01713=1057.817,-66.314,434.360,171.071,27.925,155.247
C01714=1057.824,-66.033,434.347,171.073,27.926,155.247
C01715=1057.829,-65.783,434.335,171.075,27.928,155.247
C01716=1057.836,-65.533,434.324,171.076,27.930,155.247
C01717=1057.842,-65.284,434.312,171.078,27.931,155.248
C01718=1057.848,-65.035,434.300,171.080,27.933,155.248
C01719=1057.854,-64.784,434.288,171.082,27.934,155.248
C01720=1057.861,-64.535,434.276,171.083,27.936,155.248
C01721=1057.866,-64.285,434.265,171.086,27.938,155.248
C01722=1057.872,-64.035,434.253,171.088,27.940,155.248
C01723=1057.879,-63.786,434.241,171.090,27.941,155.248
C01724=1057.885,-63.537,434.229,171.091,27.943,155.248
C01725=1057.891,-63.286,434.217,171.093,27.945,155.249
C01726=1057.897,-63.037,434.205,171.095,27.946,155.249
C01727=1057.904,-62.787,434.193,171.097,27.947,155.249
C01728=1057.910,-62.538,434.183,171.098,27.949,155.249
C01729=1057.915,-62.288,434.170,171.100,27.951,155.249
C01730=1057.922,-62.038,434.158,171.102,27.952,155.249
C01731=1057.928,-61.789,434.146,171.103,27.954,155.249
C01732=1057.934,-61.539,434.135,171.105,27.956,155.250
C01733=1057.940,-61.289,434.123,171.107,27.957,155.250
C01734=1057.947,-61.040,434.111,171.109,27.959,155.250
C01735=1057.952,-60.791,434.099,171.110,27.961,155.250
C01736=1057.959,-60.540,434.087,171.112,27.962,155.250
C01737=1057.965,-60.291,434.075,171.114,27.964,155.250
C01738=1057.971,-60.041,434.063,171.116,27.965,155.250
C01739=1057.977,-59.792,434.051,171.117,27.967,155.250
C01740=1057.984,-59.542,434.040,171.119,27.968,155.251
C01741=1057.990,-59.292,434.027,171.121,27.970,155.251
C01742=1057.996,-59.042,434.015,171.122,27.972,155.251
C01743=1058.002,-58.794,434.004,171.125,27.974,155.251
C01744=1058.008,-58.544,433.991,171.127,27.975,155.251
C01745=1058.015,-58.294,433.979,171.129,27.977,155.251
C01746=1058.020,-58.044,433.967,171.130,27.979,155.251
C01747=1058.027,-57.794,433.956,171.132,27.980,155.252
C01748=1058.033,-57.545,433.944,171.134,27.982,155.252
C01749=1058.039,-57.295,433.931,171.135,27.984,155.252
C01750=1058.046,-57.046,433.919,171.137,27.985,155.252
C01751=1058.052,-56.796,433.907,171.139,27.987,155.252
C01752=1058.058,-56.546,433.895,171.141,27.989,155.252
C01753=1058.064,-56.297,433.883,171.142,27.990,155.252
C01754=1058.071,-56.048,433.871,171.144,27.992,155.253
C01755=1058.077,-55.797,433.860,171.146,27.994,155.253
C01756=1058.083,-55.548,433.848,171.148,27.995,155.253
C01757=1058.089,-55.298,433.835,171.149,27.997,155.253
C01758=1058.096,-55.048,433.823,171.151,27.999,155.253
C01759=1058.102,-54.799,433.811,171.153,28.000,155.253
C01760=1058.108,-54.550,433.799,171.154,28.002,155.253
C01761=1058.114,-54.300,433.787,171.156,28.004,155.254
C01762=1058.120,-54.050,433.774,171.158,28.005,155.254
C01763=1058.127,-53.801,433.762,171.160,28.007,155.254
C01764=1058.134,-53.551,433.750,171.161,28.009,155.254
C01765=1058.139,-53.301,433.738,171.163,28.010,155.254
C01766=1058.146,-53.051,433.726,171.165,28.012,155.254
C01767=1058.152,-52.802,433.713,171.166,28.014,155.254
C01768=1058.159,-52.552,433.701,171.168,28.015,155.255
C01769=1058.164,-52.303,433.689,171.170,28.017,155.255
C01770=1058.171,-52.053,433.677,171.172,28.019,155.255
C01771=1058.177,-51.804,433.665,171.173,28.020,155.255
C01772=1058.183,-51.554,433.653,171.176,28.022,155.255
C01773=1058.190,-51.304,433.641,171.178,28.024,155.255
C01774=1058.196,-51.054,433.628,171.180,28.026,155.255
C01775=1058.203,-50.775,433.614,171.181,28.028,155.256
C01776=1058.210,-50.496,433.601,171.183,28.030,155.256
C01777=1058.218,-50.216,433.587,171.185,28.031,155.256
C01778=1058.224,-49.936,433.573,171.187,28.034,155.256
C01779=1058.230,-49.687,433.560,171.189,28.035,155.256
C01780=1058.236,-49.438,433.549,171.191,28.038,155.257
C01781=1058.242,-49.188,433.536,171.192,28.039,155.257
C01782=1058.248,-48.939,433.523,171.194,28.041,155.257
C01783=1058.255,-48.689,433.511,171.196,28.043,155.257
C01784=1058.261,-48.439,433.498,171.197,28.045,155.257
C01785=1058.267,-48.189,433.486,171.199,28.047,155.258
C01786=1058.273,-47.939,433.473,171.201,28.048,155.258
C01787=1058.279,-47.690,433.461,171.202,28.050,155.258
C01788=1058.285,-47.441,433.448,171.204,28.052,155.258
C01789=1058.291,-47.191,433.435,171.206,28.054,155.258
C01790=1058.297,-46.941,433.423,171.208,28.056,155.258
C01791=1058.303,-46.692,433.411,171.209,28.058,155.259
C01792=1058.309,-46.443,433.398,171.211,28.059,155.259
C01793=1058.315,-46.193,433.385,171.213,28.061,155.259
C01794=1058.321,-45.943,433.373,171.214,28.063,155.259
C01795=1058.328,-45.693,433.361,171.216,28.065,155.259
C01796=1058.334,-45.444,433.348,171.218,28.067,155.259
C01797=1058.340,-45.194,433.335,171.219,28.069,155.260
C01798=1058.346,-44.944,433.323,171.221,28.071,155.260
C01799=1058.353,-44.695,433.311,171.223,28.072,155.260
C01800=1058.359,-44.445,433.297,171.225,28.074,155.260
C01801=1058.365,-44.196,433.285,171.226,28.076,155.260
C01802=1058.371,-43.946,433.272,171.228,28.078,155.261
C01803=1058.377,-43.696,433.259,171.230,28.080,155.261
C01804=1058.383,-43.447,433.247,171.231,28.082,155.261
C01805=1058.389,-43.197,433.234,171.233,28.084,155.261
C01806=1058.396,-42.948,433.221,171.235,28.086,155.261
C01807=1058.402,-42.698,433.209,171.236,28.087,155.262
C01808=1058.407,-42.448,433.196,171.238,28.090,155.262
C01809=1058.414,-42.199,433.183,171.240,28.091,155.262
C01810=1058.420,-41.949,433.171,171.242,28.093,155.262
C01811=1058.427,-41.700,433.158,171.243,28.095,155.262
C01812=1058.432,-41.450,433.145,171.245,28.097,155.263
C01813=1058.438,-41.200,433.132,171.247,28.098,155.263
